(* CODESYS project base_elements.library
   Company: Vistaprint
   Version: 0.0.0.1
   Title: Base_Elements

Project tree, tasks and I/O mapping:
  libraries: Base_PLC, 0.3.2.0 (Vistaprint); Tc2_EtherCAT, 3.3.0.0 (Beckhoff Automation GmbH); Tc2_SerialCom, 3.3.0.0 (Beckhoff Automation GmbH); Tc2_Standard, * (Beckhoff Automation GmbH); Tc2_System, * (Beckhoff Automation GmbH); Tc2_Utilities, 3.3.0.0 (Beckhoff Automation GmbH); Tc3_Interfaces, * (Beckhoff Automation GmbH); Tc3_Module, * (Beckhoff Automation GmbH)
  POUs/
    Controller/
      Driver/
        RFD (RFID Driver)/
          data type E_Typ_Baudrate
          data type E_Typ_Ftim
          function block FB_Com_3964R [ST]
          function block FB_ExCom [ST]
          function FB_HEXSTRING_TO_ULINT [ST]
          function block FB_RFD [ST]: CtrlInit, CycleEndDuty, CycleStartDuty, FB_init, getCmdState, getSIf, sta_CheckBusy, sta_Error, sta_MDSBusy, sta_Off, sta_OffBusy, sta_PowerOnBusy, sta_ReadBusy, sta_SLGBusy, sta_TagInitBusy, sta_WaitForJob, sta_WriteBusy, StateMachine, StateMachine_Service
          function block FB_RFR [ST]: CtrlInit, CycleEndDuty, CycleStartDuty, FB_init, getCmdState, getSIf, sta_Error, sta_PowerOnBusy, sta_WaitForJob, StateMachine, StateMachine_Service
          global variables RFD_Cmd
          global variables RFD_Constants
          data type T_RFD
          data type T_RFD_Cfg
          data type T_RFD_Cur
          data type T_RFD_Error
          data type T_RFD_MDS_Diagnose
          data type T_RFD_MDS_State
          data type T_RFD_SLG_Diagnose
          data type T_RFD_SLG_State
          data type T_RFD_StateMachine
          data type T_RFD_Status
          data type T_StateWord
      Lvl0/
        RFW (RFID Reader-Writer)/
          data type E_Typ_RFW
          function block FB_DtChnToLine_NewRFID [ST]: Creat
          function block FB_RFW [ST]: Always, FB_init, getCmdState, getCtrlSIf, IoInBridge, IoOutBridge, sta_ERROR, sta_OFF, sta_OFFBusy, sta_PON, sta_PONBusy, sta_READ, sta_READBusy, sta_RUN, sta_RUNbusy, sta_WRITE, sta_WRITEBusy, StateMachine
          function FB_ULINT_TO_HEXSTRING [ST]
          global variables RFID_Data
          global variables RFW_CmdState
          data type T_Ctrl_SIf_RFW
          data type T_Ctrl_SIf_RFW_Cfg
          data type T_Ctrl_SIf_RFW_Cur
          data type T_Ctrl_SIf_RFW_DtChnToLine
          data type T_Ctrl_SIf_RFW_In
          data type T_Ctrl_SIf_RFW_Out
          data type T_Ctrl_SIf_RFW_Par
          data type T_NewRFID_DtChn
          data type T_RFW
      Lvl1/
      Lvl2/
      Lvl3/
    Utility Functions/
  Version/
    global variables Global_Version
*)

// POUs/Controller/Driver/RFD (RFID Driver)/E_Typ_Baudrate
TYPE E_Typ_Baudrate :
(
	baud_2400 := 4,
	baud_4800 := 5,
	baud_9600 := 6,
	baud_19200 := 7,
	baud_38400 := 8,
	baud_57600 := 9,
	baud_115200 := 10
);
END_TYPE

// POUs/Controller/Driver/RFD (RFID Driver)/E_Typ_Ftim
TYPE E_Typ_Ftim :
(
	/// Setting for air interface
	RF300 := 0,
	ISO_generall := 1,
	ISO_infineon := 3,
	ISO_Fujitsu := 4,
	ISO_NXP := 5,
	ISO_TI := 6,
	ISO_ST := 7,
	Max_E_Typ_Ftim
);
END_TYPE

// POUs/Controller/Driver/RFD (RFID Driver)/T_RFD
TYPE T_RFD :
STRUCT
	strState: STRING;
	strCmd: STRING;
	intCmd: INT;
	intServiceCmd: INT;
	stStatus: T_RFD_Status;
	stCfg: T_RFD_Cfg;
	stCur: T_RFD_Cur;
	stErr: T_RFD_Error;
END_STRUCT
END_TYPE

// POUs/Controller/Driver/RFD (RFID Driver)/T_RFD_Cfg
TYPE T_RFD_Cfg :
STRUCT
	bolSimulation: BOOL;
	eTyp: E_Typ_RFW;
	/// Reset parameter value
	usiResetParameter: USINT := 2#101010;
	/// Setting of the Air interface
	usiFtimSetting: E_Typ_Ftim;
	/// Reset option1 value
	usiResetOption1: USINT := 2#10;
	/// Set Baudrate
	uinBaudrate: USINT;
	/// Set Communikationsettings
	uinComSettings: USINT;
	/// Net ID oft EtherCat Master
	stNetId: TC2_SYSTEM.T_AmsNetID;
	/// Port Number of EtherCat Slave Comunication Module
	uinSlaveAddr: UINT;
	/// CoE Object Index for Communication Settings
	uinCoeIndexComSettings: WORD := 16#8000;
	/// CoE Object SubIndex for Baudrate
	usiCoeSubindexComBaudrate: BYTE := 16#11;
	/// CoE Object SubIndex for Dataframe
	usiCoeSubindexComDataframe: BYTE := 16#15;
	/// Retry Job to RFID Reader
	udiRetry: UDINT := 10;
	//////////////////////////////////////////////////
	/// Reset Memory 00=RAM, 01=remanent
	usiMemory: USINT := 0;
	/// Scan Mode 00= Continous Read; 01=Single Read
	usiScanMode: USINT := 1;
	/// Lock Time in ms
	uinLockTime_ms: UINT := 5000;
END_STRUCT
END_TYPE

// POUs/Controller/Driver/RFD (RFID Driver)/T_RFD_Cur
TYPE T_RFD_Cur :
STRUCT
	/// Pointer to Received Data Array
	pData: POINTER TO ARRAY[0..255] OF BYTE;
	/// Startadress to Read/Write at the data Array Element
	uinAdressData: UINT;
	/// Startadress to Read/Write at the Tag
	uinAdressTag: UINT;
	/// Number of bytes to Read/Write
	usiCount: USINT;
END_STRUCT
END_TYPE

// POUs/Controller/Driver/RFD (RFID Driver)/T_RFD_Error
TYPE T_RFD_Error :
STRUCT
	/// Reset failure
	bolErrAck: BOOL;
	/// atleast one failure active
	bolErrorActive: BOOL;
	/// error at communication card
	bolComError: BOOL;
	bolProtcolError: BOOL;
	/// Error with RF ID Tag
	bolRFIDError: BOOL;
	/// Error at setting of the communication Card (SDO Write)
	bolSDOError: BOOL;
	/// information to Communication Card error
	udiErrorID: UDINT;
END_STRUCT
END_TYPE

// POUs/Controller/Driver/RFD (RFID Driver)/T_RFD_MDS_Diagnose
TYPE T_RFD_MDS_Diagnose :
STRUCT
	/// Power flux density: as smaller the value, as higher the field intensity
	usiLFD: USINT;
	/// Errorcounter inactive mode
	usiFZP: USINT;
	/// Errorcounter active: CRC or signature errors
	usiFZA: USINT;
	/// Presence time of tag, resolution in 9.7ms
	usiANWZ: USINT;
END_STRUCT
END_TYPE

// POUs/Controller/Driver/RFD (RFID Driver)/T_RFD_MDS_State
TYPE T_RFD_MDS_State :
STRUCT
	/// MDS Type 1=no FRAM; 2=8k FRAM; 3=32k FRAM; 4=64k FRAM; 5=128k FRAM; 6=256k FRAM
	bytMDSType: BYTE;
	/// Lock bit registers (lock state)
	bytLockState: BYTE;
	/// MDS Version
	bytVersion: BYTE;
	/// Memory Size
	worMemSize: WORD;
	/// Blocksize in Byte
	bytBlockSize: BYTE;
	/// Value of memory Blocks
	bytBlockNo: BYTE;
END_STRUCT
END_TYPE

// POUs/Controller/Driver/RFD (RFID Driver)/T_RFD_SLG_Diagnose
TYPE T_RFD_SLG_Diagnose :
STRUCT
	/// Mode SLG Diagnose
	usiS_Info: USINT;
	/// Errorcounter inactive mode
	usiFZP: USINT;
	/// Counter abort
	usiABZ: USINT;
	/// Errorcounter code errors
	usiCFZ: USINT;
	/// Errorcounter signature errors
	usiSFZ: USINT;
	/// Errorcounter CRC
	usiCRCFZ: USINT;
	/// Actual command state
	usiBSTAT: USINT;
	/// Counter interface errors to host (Parity, BCC, Frame)
	usiASMFZ: USINT;
END_STRUCT
END_TYPE

// POUs/Controller/Driver/RFD (RFID Driver)/T_RFD_SLG_State
TYPE T_RFD_SLG_State :
STRUCT
	/// HW Type of SLG  0=RF310R RF340R RF350R (-xAA10); 1=RF380R (-3AA10); 2=RF310R(-1AB10); 3=RF380R (-3AB10); 4=RF340R RF350R (-2AB10,-4AB10)
	bytHWType: BYTE;
	/// HW Version
	worHWVersion: WORD;
	/// Loading Version
	worURLVersion: WORD;
	/// FW Type
	bytFWType: BYTE;
	/// FW Version
	worFWVersion: WORD;
	/// Driver Type 1=3964R
	bytDriverType: BYTE;
	/// Driver Version
	worDriverVersion: WORD;
	/// Communication port 1=RS422, 2=RS232
	bytComm: BYTE;
	/// Communication Baud rate 1=19.2kBaud; 3=57.6kBaud; 5=115.2kBaud
	bytBaud: BYTE;
	/// sending power (only RF380R) 0=standard; 2=0.5W; 3=0.75W; 4=1W; 5=1.25W (default); 6=1.5W; 7=1.75W; 8=2W
	bytPower: BYTE;
	/// Number of maximal tags in the field
	bytMtag: BYTE;
	/// air interface 0=RF300; 1=ISO generall; 3=ISO infineon Chip; 4=ISO Fujitsu; 5=ISO NXP; 6=ISO TI; 7=ISO ST
	bytFtim: BYTE;
	/// State antenna 1=ON; 2=OFF
	bytAntenna: BYTE;
	/// Tag presence 0=No presence; 1=prexence
	bytPresence: BYTE;
END_STRUCT
END_TYPE

// POUs/Controller/Driver/RFD (RFID Driver)/T_RFD_StateMachine
TYPE T_RFD_StateMachine :
STRUCT
	///actual state
	intState: INT;
	///state of last cycle
	intStateLastCycle: INT;
	///save history backup p.e. in ERROR state
	intStateHistory: INT;
	///set state for next cycle
	intStateNext: INT;
	///Time in this State
	udiTimeInState_ms: UDINT;
END_STRUCT
END_TYPE

// POUs/Controller/Driver/RFD (RFID Driver)/T_RFD_Status
TYPE T_RFD_Status :
STRUCT
	/// 1 = Antenna is initialized  
	bolStartupOk: BOOL;
	/// 1 = Antenna is initialized  
	bolInitOk: BOOL;
	/// 1 = Antenna is on 
	bolOn: BOOL;
	/// 1 = tag is present  
	bolPresent: BOOL;
	/// 1 = Communication to SLG is OK  
	bolL_UEB: BOOL;
	/// SLG State only actual on demand 
	stSLG_State: T_RFD_SLG_State;
	/// SLG Diagnose only actual on demand 
	stSLG_Diag: T_RFD_SLG_Diagnose;
	/// SLG State only actual on demand  
	stMDS_State: T_RFD_MDS_State;
	/// SLG Diagnose only actual on demand  
	stMDS_Diag: T_RFD_MDS_Diagnose;
	/// Tag ID
	abyteUID: ARRAY[0..7] OF BYTE;
END_STRUCT
END_TYPE

// POUs/Controller/Driver/RFD (RFID Driver)/T_StateWord
TYPE T_StateWord :
STRUCT
	///Acknowledge the datachange of this Command bit
	bolTransmitAccepted: BOOL;
	///New Datat at the input
	bolReceiveRequest: BOOL;
	///0=Ready for Data exchange; 1=initialisation of the clam
	bolInputAccepted: BOOL;
	///Input Buffer is full, all new arriveing data lost
	bolBufferFull: BOOL;
	///Parity Error occured
	bolParityErr: BOOL;
	///Framing Error occured
	bolFramingErr: BOOL;
	///Overrun Error occured
	bolOverrunErr: BOOL;
	///Amounth of the reached Input Bytes
	usiInLenght: USINT;
END_STRUCT
END_TYPE

// POUs/Controller/Lvl0/RFW (RFID Reader-Writer)/E_Typ_RFW
TYPE E_Typ_RFW :
(
	/// RF310
	RF310R := 0,
	/// RF382R
	RF382R := 1,
	Max_E_Typ_CYL
);
END_TYPE

// POUs/Controller/Lvl0/RFW (RFID Reader-Writer)/T_Ctrl_SIf_RFW
TYPE T_Ctrl_SIf_RFW :
STRUCT
	///configuration
	Cfg: T_Ctrl_SIf_RFW_Cfg;
	///parameter
	Par: T_Ctrl_SIf_RFW_Par;
	///current values
	Cur: T_Ctrl_SIf_RFW_Cur;
	///io input
	In: T_Ctrl_SIf_RFW_In;
	///io output
	Out: T_Ctrl_SIf_RFW_Out;
	///alarm number used in this controller
	Alm: ARRAY[1..5] OF T_Ctrl_Alm;
END_STRUCT
END_TYPE

// POUs/Controller/Lvl0/RFW (RFID Reader-Writer)/T_Ctrl_SIf_RFW_Cfg
TYPE T_Ctrl_SIf_RFW_Cfg :
STRUCT
	eTyp: E_Typ_RFW;
	/// Get automatically the Tray ID too 
	bolGetTrayIDAuto: BOOL;
	/// Net ID oft EtherCat Master
	stNetId: TC2_SYSTEM.T_AmsNetID;
	/// Port Number of EtherCat Slave Comunication Module
	uinSlaveAddr: UINT;
END_STRUCT
END_TYPE

// POUs/Controller/Lvl0/RFW (RFID Reader-Writer)/T_Ctrl_SIf_RFW_Cur
TYPE T_Ctrl_SIf_RFW_Cur :
STRUCT
	/// 1 = tag is present  
	bolPresent: BOOL;
	/// Data to read / write
	abytData: ARRAY[0..255] OF BYTE;
	/// Data in Structure
	stData: T_RFW;
	/// Job information, what data read or write
	dwoJob: DWORD;
END_STRUCT
END_TYPE

// POUs/Controller/Lvl0/RFW (RFID Reader-Writer)/T_Ctrl_SIf_RFW_DtChnToLine
TYPE T_Ctrl_SIf_RFW_DtChnToLine :
STRUCT
	stNewRfid: T_NewRFID_DtChn;
END_STRUCT
END_TYPE

// POUs/Controller/Lvl0/RFW (RFID Reader-Writer)/T_Ctrl_SIf_RFW_In
TYPE T_Ctrl_SIf_RFW_In :
STRUCT
END_STRUCT
END_TYPE

// POUs/Controller/Lvl0/RFW (RFID Reader-Writer)/T_Ctrl_SIf_RFW_Out
TYPE T_Ctrl_SIf_RFW_Out :
STRUCT
END_STRUCT
END_TYPE

// POUs/Controller/Lvl0/RFW (RFID Reader-Writer)/T_Ctrl_SIf_RFW_Par
TYPE T_Ctrl_SIf_RFW_Par :
STRUCT
	///[ms] until failure to long time for read
	udiReadTime_ms: UDINT;
	///[ms] until failure to long time for write
	udiWriteTime_ms: UDINT;
END_STRUCT
END_TYPE

// POUs/Controller/Lvl0/RFW (RFID Reader-Writer)/T_NewRFID_DtChn
TYPE T_NewRFID_DtChn :
STRUCT
	// new RF ID
	strID: STRING;			// configurable if Tag or Tray ID
	uliTagID: ULINT;
	dtTimestamp: DT;
	intDataState: INT;	
END_STRUCT
END_TYPE

// POUs/Controller/Lvl0/RFW (RFID Reader-Writer)/T_RFW
TYPE T_RFW :
STRUCT
	///	Repeteition ID			Identifies the try number in the sequence	
	usiRepetitionID: USINT;
	///	Workstation		2 workstations in the cell	1 BIT	0: Workstation1, 2: Workstation2
	bolWorkstation2: BOOL;
	///usiProductID : USINT;				// 	The product ID bits 1 to 5 are indeed not used. Mail T.Bosgiraud 11.6.2013 Product type	Max number of product types = 32	5 bits,	product ID (bits 1 to 5), 
	bolDeleteFileAfterPrint: BOOL;
	/// 	1 means that the image has been printed without problem.
	bolPrintOk: BOOL;
	///	0: Use the bottom of the tray as basis and add Offset
	bolHeightUseMeasure: BOOL;
	///	Email 1.06.2013 Berk “Use measured height=1”, the actual measurement of the  laser plus any offsets programmed into the tray are used to adjust the lifting height
	///	1: Use the printable product surface as basis and add Offset to the measured height
	usiHeightOffset: USINT;
	/// 	“Offset +/-” = 1 means that the printable surface OF the item will go further away FROM the print head.
	bolHeightOffsetSignMinus: BOOL;
	/// 	“Offset +/-” = 0 (default value) means that the printable surface of the item will come closer to the print head
	bolIonizer: BOOL;
	/// 	Pre-treatment	Plasma 0: Plasma off, 1: Level 1 ..3:Level3
	usiPlasmaLevel: USINT;
	/// 	Print numbers 1 means that the image needs to be printed twice on the products
	bolPrintPass: BOOL;
	/// 	1 means that the nozzle check pattern has to be printed onto the products.
	bolNozzleCheck: BOOL;
	///	1 means that the alignment check pattern has to be printed onto the products.
	bolAligneCheck: BOOL;
	///	UV-pinning intensity 0: Level1 ... 15: Level16
	usiUVPinningLevel: USINT;
	///	UV-lamp intensity 0: Level1 ... 15: Level16
	usiUVLampLevel: USINT;
	/// p.e.: 268205625-3.pdf -> The file name sent by VIPER to the printer and to the conveyor is made out of 64 bits
	strFileName: STRING;
	/// The RFID divides the rest of the name (268205625-3) as 8 successive bytes arranged as follows:
	///	-	Byte 7 (RFID byte 0Dhex) to byte 1 (RFID byte 07hex) express the number before the hyphen sign (in this case 268205625)
	///	-	Byte 0 (RFID byte 06hex) expresses the number after the hyphen sign (in this case 3).
	bolBrush: BOOL;
	///	1: use second brush means that the brush has TO be used FOR the considered tray
	bolBrushClean: BOOL;
	///	“Brush Fans”=1 means that the fans have to be used for the considered tray
	bolBrushFans: BOOL;
	///	“Gutter Clean”=1 means that the tray is running for gutter cleaning purposes.
	bolGutterClean: BOOL;
	/// 	This bit tells whether the tray is a regular production tray or a special tray (nozzle check, alignment...).
	bolSpecialTray: BOOL;
	/// 	Byte 0-13	->9999999999999	
	strTrayID: STRING;
	/// 	Byte 0-13	->9999999999999	
	strTagID: STRING;
	uliTagID: ULINT;
END_STRUCT
END_TYPE

// POUs/Controller/Driver/RFD (RFID Driver)/RFD_Cmd
VAR_GLOBAL CONSTANT
	/// ctrl state definitions
	/// Error
	cRFD_STA_Error: INT := 256;
	/// Power On
	cRFD_STA_PowerOnBusy: INT := 999;
	cRFD_STA_WaitForJob: INT := 1002;
	/// RESET Reader 
	cRFD_STA_ResetBusy: INT := 1003;
	/// Turn Off antenna 
	cRFD_STA_OffBusy: INT := 1007;
	cRFD_STA_Off: INT := 1008;
	/// Write Data to Tag 
	cRFD_STA_WriteBusy: INT := 1009;
	/// Read Data from Tag 
	cRFD_STA_ReadBusy: INT := 1011;
	/// Tag initialisation 
	cRFD_STA_TagInitBusy: INT := 1013;
	/// Check connection to antenna
	cRFD_STA_CheckBusy: INT := 1017;
	/// Service function read MDS-State (State of the near Tag)
	cRFD_STA_MDSBusy: INT := 1019;
	/// Service function read SLG State (State of the antenna)
	cRFD_STA_SLGBusy: INT := 1021;
	/// ctrl commands definitions
	/// specific commands >200 - every command has to be a even number
	cRFD_CMD_DONE: INT := -1;
	/// Switch controller on 
	cRFD_CMD_CTRL_ON: INT := 1000;
	/// Switch controller off 
	cRFD_CMD_CTRL_OFF: INT := 1006;
	/// Write Data to Tag 
	cRFD_CMD_Write: INT := 1010;
	/// Read Data from Tag 
	cRFD_CMD_Read: INT := 1012;
	/// Check connection to antenna 
	cRFD_CMD_Check: INT := 1018;
	/// Service function read MDS-State (State of the near Tag)
	cRFD_CMD_MDS: INT := 1020;
	/// Service function read SLG State (State of the antenna)
	cRFD_CMD_SLG: INT := 1022;
	/// Sub States
	/// Power On Busy
	cRFD_SUB_SetBaudrate: INT := 2001;
	/// Set Communication Settings
	cRFD_SUB_SetComSettings: INT := 2002;
	///  Clear Buffer
	cRFD_SUB_ClearBuffer: INT := 2003;
	/// Initialisation String sending
	cRFD_SUB_InitString: INT := 2004;
	///  Check Power On State
	cRFD_SUB_CheckPon: INT := 2005;
	/// OFF Busy
	cRFD_SUB_Prepare: INT := 2010;
	/// Data send
	cRFD_SUB_SendBusy: INT := 2011;
	/// Wait Answer
	cRFD_SUB_WaitAnswer: INT := 2012;
	/// SLG Write Mode 1
	cRFD_SUB_Write1: INT := 2020;
	/// SLG Wait Mode 1
	cRFD_SUB_Wait1: INT := 2021;
	/// SLG Write Mode 6
	cRFD_SUB_Write6: INT := 2022;
	/// SLG Wait Mode 6
	cRFD_SUB_Wait6: INT := 2023;
	///  Substates finished
	cRFD_SUB_SubStatesEnd: INT := 2100;
END_VAR

// POUs/Controller/Driver/RFD (RFID Driver)/RFD_Constants
VAR_GLOBAL
END_VAR

// POUs/Controller/Lvl0/RFW (RFID Reader-Writer)/RFID_Data
VAR_GLOBAL CONSTANT
	/// RFID Data connection
	/// See RFID Specification
	/// Defines the Start Adress and the lengh of the Data in the RF ID Tag
	/// Every DoubleWord has to Words, Higher is lengh, lower word is Startadress
	/// Example	
	/// 16#010005 => Startadress 5 Byte 1 => UV Settings
	cRFID_RepetionID: DWORD := 16#10101;
	cRFID_TrayInfo: DWORD := 16#10102;
	cRFID_HeighOfTray: DWORD := 16#10103;
	cRFID_Pretreatment: DWORD := 16#10104;
	cRFID_UVcuring: DWORD := 16#10105;
	cRFID_Filename: DWORD := 16#80106;
	cRFID_Brush: DWORD := 16#1010E;
	cRFID_TrayID: DWORD := 16#E0000;
	cRFID_TagID: DWORD := 16#8FFF0;
	cRFID_AllData: DWORD := 16#F0100;
END_VAR

// POUs/Controller/Lvl0/RFW (RFID Reader-Writer)/RFW_CmdState
VAR_GLOBAL CONSTANT
	///ctrl commands definitions
	///specific commands >200 - every command has to be a even number
	cCMD_READ: INT := 202;
	cCMD_WRITE: INT := 204;
	///ctrl specific states definitions
	cSTA_READBusy: INT := 201;
	cSTA_READ: INT := cCMD_READ;
	cSTA_WRITEBusy: INT := 203;
	cSTA_WRITE: INT := cCMD_WRITE;
END_VAR

// Version/Global_Version
// This function has been automatically generated from the project information.
VAR_GLOBAL CONSTANT
	{attribute 'const_non_replaced'}
	stLibVersion_Base_Elements : ST_LibVersion := (iMajor := 0, iMinor := 0, iBuild := 0, iRevision := 1, sVersion := '0.0.0.1');
END_VAR

// POUs/Controller/Driver/RFD (RFID Driver)/FB_Com_3964R
FUNCTION_BLOCK FB_Com_3964R
VAR_INPUT
	/// Pointer to Received Data Array
	In_pRxData: POINTER TO ARRAY[0..255] OF BYTE;
	/// Pointer to Sending Data Array
	In_pTxData: POINTER TO ARRAY[0..255] OF BYTE;
	/// Amounth of sending data
	In_udiTxCount: UDINT;
	/// Error Acknowledge 
	In_bolErrorAck: BOOL;
END_VAR
VAR_IN_OUT
	/// Command to send Data 1=command; 0=Done
	InOut_bolSend: BOOL;
	/// Command Data received 1=received; 0=Done=Ready for next Data
	InOut_bolRec: BOOL;
END_VAR
VAR_OUTPUT
	/// Amounth of received data
	Out_udiRxCount: UDINT;
	/// Serial interface communication error
	Out_bolComError: BOOL;
	/// Error in protocoll procedure
	Out_bolProtocolErr: BOOL;
	/// Error information to master
	Out_udiErrorCode: UDINT;
END_VAR
VAR
	In_stEL6inData AT %I*: TC2_SERIALCOM.EL6inData22B;
	Out_stEL6outData AT %Q*: TC2_SERIALCOM.EL6outData22B;
	/// Internal Variables
	udiI: UDINT;
	/// Local variable for loops
	udiK: UDINT;
	/// Internal Error Reset
	bolIntReset: BOOL;
	/// Count call trials
	uinCountCall: UINT;
	/// Count call Retrys
	uinCountRetry: UINT;
	/// Temporary value for cecking the sum
	bytCheckValue: BYTE;
	/// Antenna is initializied, until it is not initializied, it send 16#02 in all possible baudrates
	bolSLGInitialized: BOOL := FALSE;
	/// Check Timeout
	bolTimeout: BOOL;
	/// Check Timeout
	bolWait: BOOL;
	/// Send NAK needed
	bolSendNAK: BOOL;
	/// Receive Wait signs
	timWaitReceive: TIME := TIME#5ms;
	/// Receive Wait signs
	timWaitAck: TIME := TIME#400ms;
	/// Sign delay time
	timZVZ: TIME := TIME#45ms;
	/// Time ACK delay
	timQVZ: TIME := TIME#145ms;
	/// Initialisation of the HW card
	bolInitRequest: BOOL;
	/// Setting of the HW Card
	bolSendContinious: BOOL;
	/// Priority at RFID
	bolPriority: BOOL;
	/// Send DLE doubletimes
	bolDLEDouble: BOOL;
	/// New data received
	bolComDataReceived: BOOL;
	/// receiving busy
	bolComRecBusy: BOOL;
	/// Received Data
	udiComSizeReceiveData: UDINT;
	/// Sending busy
	bolComSendBusy: BOOL;
	/// Error at serial line control
	bolErrSerialLineControl: BOOL;
	/// Error at serial line control
	stErrSerialLineControl: ComError_t;
	/// Error at serial line  receiving data
	bolErrReceive: BOOL;
	/// Error at serial line  receiving data
	stErrReceive: ComError_t;
	/// Error at serial line sending data
	bolErrSend: BOOL;
	/// Error at serial line sending data
	stErrSend: ComError_t;
	/// Define Buffer for preparations
	aRxData: ARRAY[0..255] OF BYTE;
	aTxData: ARRAY[0..255] OF BYTE;
	/// Define Buffer for Funciton
	stRxBuffer: TC2_SERIALCOM.ComBuffer;
	/// Transmit data buffer; used with all receive function blocks 
	stTxBuffer: TC2_SERIALCOM.ComBuffer;
	/// Sub Statemachine
	intState: INT := 0;
	intStateOld: INT := 0;
	udiStateLoop: UDINT;
	a_intStateHist: ARRAY[0..9] OF INT;
	udiStateDebug: UDINT;
	udiStateDebugMax: UDINT;
	/// Function for serial communication
	fbSerialLineControl: TC2_SERIALCOM.SerialLineControl;
	fbSerialReceiveData: TC2_SERIALCOM.ReceiveData;
	fbSerialSendData: TC2_SERIALCOM.SendData;
	fbSerialClearComBuffer: TC2_SERIALCOM.ClearComBuffer;
	fbTon: TC2_STANDARD.TON;
	fbWait: TC2_STANDARD.TON;
	fbZVZ: TC2_STANDARD.TON;
	fbQVZ: TC2_STANDARD.TON;
	fbPriority: TC2_STANDARD.TON;
END_VAR
VAR CONSTANT
	cSTX: USINT := 16#2;
	cDLE: USINT := 16#10;
	cETX: USINT := 16#3;
	cNAK: USINT := 16#15;
	/// Startup
	cRFD_3964_Start: INT := 2500;
	/// Startup
	cRFD_3964_Init: INT := 2501;
	/// Wait for Job
	cRFD_3964_Wait: INT := 2502;
	/// Read recived sign
	cRFD_3964_RxRead: INT := 2504;
	/// Ackn. receiving ready
	cRFD_3964_RxReadRdy: INT := 2506;
	/// Recive Data
	cRFD_3964_RxData: INT := 2508;
	/// Achn. received Data
	cRFD_3964_RxCheckData: INT := 2510;
	/// Send Ack to Slave
	cRFD_3964_RxAck: INT := 2512;
	/// Send Ack to Slave
	cRFD_3964_RxAck2: INT := 2514;
	/// Send Request to Slave
	cRFD_3964_TxRequest: INT := 2550;
	/// Send Wait answer
	cRFD_3964_TxWait: INT := 2552;
	/// Send Data
	cRFD_3964_TxSend: INT := 2554;
	/// Send Wait for Ack
	cRFD_3964_TxAck: INT := 2556;
	/// Error
	cRFD_3964_Error: INT := 2580;
END_VAR

(*__________________________________________________________________________________________________
¦	
¦	Vistaprint Schweiz GmbH
¦	CH - 8401 Winterthur
¦
¦	www.vistaprint.ch - info@vistaprint.ch
¦___________________________________________________________________________________________________

Function desription:
Driver for communication protocoll 3964R
Description in Siemens manual from CP341, A5E02191070-03


History:
Version		Date			Author		Comment
---------------------------------------------------------------------------------------------------
0.00.1		23.07.2013		AVME/PRE	Start history
___________________________________________________________________________________________________*)

// Always
fbSerialLineControl(
	Mode:= TC2_SERIALCOM.ComSerialLineMode_t.SERIALLINEMODE_EL6_22B, 
	pComIn:= ADR(In_stEL6inData), 
	pComOut:= ADR(Out_stEL6outData), 
	SizeComIn:= SIZEOF(In_stEL6inData), 
	Error=> bolErrSerialLineControl, 
	ErrorID=> stErrSerialLineControl, 
	TxBuffer:= stTxBuffer, 
	RxBuffer:= stRxBuffer);
	
// Check timers
IF intState >= cRFD_3964_Wait THEN
	fbZVZ(PT:= timZVZ);
	fbQVZ(PT:= timQVZ);
	fbWait(PT:= timWaitAck);

	// Check priority
	fbPriority(IN:= bolPriority, PT:=timWaitAck);
	IF (fbPriority.Q = TRUE) THEN
		bolPriority := FALSE;
	END_IF

END_IF
		
// Startup set correct Step
IF intState < cRFD_3964_Start THEN
	intState := cRFD_3964_Start;
END_IF

// State Machine
CASE intState OF
	cRFD_3964_Start:
		// Clear Buffer
		FOR udiI := 0 TO SIZEOF(aRxData)-1 DO
			aRxData[udiI] := 0;
			aTxData[udiI] := 0;
		END_FOR
		bolSLGInitialized := FALSE;
		
		// Clear counters
		uinCountCall := 0;
		uinCountRetry := 0;
		
		bolInitRequest := FALSE;
		bolSendContinious := FALSE;
		
		
		// Next State
		IF (bolErrSerialLineControl = FALSE) AND (bolTimeout=TRUE) THEN
			intState := cRFD_3964_Init;
		ELSIF (bolErrSerialLineControl = TRUE) THEN
			intState := cRFD_3964_Error;
		END_IF

	// Wait for a job or received Data //	
	cRFD_3964_Init:	
		bolInitRequest := TRUE;
		
		IF (bolErrSerialLineControl = FALSE) AND ((In_stEL6inData.Status.2 = TRUE) OR (bolTimeout=TRUE)) THEN	// Initialisation Done  OR (bolTimeout=TRUE)
			intState := cRFD_3964_Wait;
		ELSIF (bolErrSerialLineControl = TRUE) THEN
			intState := cRFD_3964_Error;
		END_IF
	
	// Wait for a job or received Data //	
	cRFD_3964_Wait:	
		bolInitRequest := FALSE;
		bolSendNAK := FALSE;
		fbZVZ.IN := FALSE;
		fbQVZ.IN := FALSE;
		fbWait.IN := FALSE;
		
		fbSerialReceiveData(
		//	pPrefix:= , // Not used because no prefix in telegram
			LenPrefix:= 0, 
		//	pSuffix:= , // Not used because no suffix in telegram
			LenSuffix:= 0, 
			pReceiveData:= ADR(aRxData), 
			SizeReceiveData:= 255, 
			Timeout:= timWaitReceive, 
		//	Reset:= , 
			DataReceived=> bolComDataReceived, 
			busy=> bolComRecBusy, 
			Error=> stErrReceive, 
			RxTimeout=> bolErrReceive, 
			LenReceiveData=> udiComSizeReceiveData, 
			RXbuffer:= stRxBuffer);
		
		//Check if Data is received
		IF bolComDataReceived = TRUE THEN
			intState := cRFD_3964_RxRead;
		ELSIF (InOut_bolSend = TRUE) AND (bolPriority = FALSE) THEN
			intState := cRFD_3964_TxRequest;
		END_IF
			
	// Read first signs if new data sending needed //	
	cRFD_3964_RxRead: 
		// Check reached Sign
		// Send ready for reach Data if STX is send and Buffer is ready to use
		fbWait.IN := TRUE;
		IF (((aRxData[0] = cSTX) OR (bolSLGInitialized = FALSE))  AND (InOut_bolRec = FALSE)) THEN 
			aTxData[0] := cDLE;
		ELSE
			aTxData[0] := cNAK;
		END_IF
		
		IF ((fbWait.Q = FALSE) OR (InOut_bolRec = TRUE)) THEN
			intState := cRFD_3964_RxReadRdy; 
			fbWait.IN := FALSE; 
		END_IF
		
	// Send Feedback //		
	cRFD_3964_RxReadRdy:
		fbZVZ.IN := TRUE; 

		IF fbZVZ.Q = TRUE THEN
			fbSerialSendData(
				pSendData:= ADR(aTxData), 
				Length:= 1, 
				Busy=> bolComSendBusy, 
				Error=> stErrSend, 
				TXbuffer:= stTxBuffer);
				bolSendContinious := TRUE;
		END_IF
			
		// Check transition
		IF (bolComSendBusy = FALSE) AND (bolSLGInitialized = TRUE) AND (fbZVZ.Q = TRUE) THEN		// AND (stErrSend = 0)
			IF (aTxData[0] = cDLE) THEN
				intState := cRFD_3964_RxData;
			ELSE
				intState := cRFD_3964_Wait;
			END_IF
		ELSIF ((bolComSendBusy = TRUE) OR (bolTimeout = TRUE)) AND (uinCountCall < 10) AND (fbZVZ.Q = TRUE) THEN
			uinCountCall := uinCountCall + 1;
			intState := cRFD_3964_Wait;
		ELSIF ((bolComSendBusy = TRUE) OR (bolTimeout = TRUE)) AND (fbZVZ.Q = TRUE) THEN
			bolSendNAK := TRUE;
			intState := cRFD_3964_Error;
		END_IF
		
	// Read Data //	
	cRFD_3964_RxData:
		fbZVZ.IN := FALSE; 
		fbSerialReceiveData(
		//	pPrefix:= , // Not used because no prefix in telegram
			LenPrefix:= 0, 
		//	pSuffix:= , // Not used because no suffix in telegram
			LenSuffix:= 0, 
			pReceiveData:= ADR(aRxData), 
			SizeReceiveData:= 255, 
			Timeout:= timWaitReceive, 
		//	Reset:= , 
			DataReceived=> bolComDataReceived, 
			busy=> bolComRecBusy, 
			Error=> stErrReceive, 
			RxTimeout=> bolErrReceive, 
			LenReceiveData=> udiComSizeReceiveData, 
			RXbuffer:= stRxBuffer);
				
		IF (bolComDataReceived = TRUE) AND (bolComRecBusy = FALSE) AND (udiComSizeReceiveData <= 255)  THEN
			intState := cRFD_3964_RxCheckData;
		ELSIF ((bolTimeout = TRUE) OR (udiComSizeReceiveData > 255)) THEN	 // OR (stErrReceive <> 0)
			bolSendNAK := TRUE;
			IF (uinCountCall < 10) THEN
				uinCountCall := uinCountCall + 1;
				intState := cRFD_3964_RxAck;
			ELSE
				intState := cRFD_3964_Error;
			END_IF
		END_IF
	
	// Check Received Data //	
	cRFD_3964_RxCheckData:
		//minimal 1 Byte, ETX and BCC   	ETX is last sign for BCC					DLE is last sign for ETX
		IF (udiComSizeReceiveData >= 4) THEN
			IF ((aRxData[udiComSizeReceiveData-2] = cETX) AND (aRxData[udiComSizeReceiveData-3] = cDLE)) THEN
				// Check BCC
				bytCheckValue := aRxData[0] XOR aRxData[1];
				FOR udiI := 2 TO  (udiComSizeReceiveData-2) DO
					bytCheckValue := bytCheckValue XOR aRxData[udiI];
				END_FOR
				
				IF (bytCheckValue = aRxData[udiComSizeReceiveData-1]) THEN //BCC OK
					// Copy Data
					FOR udiI := 0 TO (SIZEOF(aRxData)-1) DO
						In_pRxData^[udiI] := 0;
					END_FOR
					udiK := 0;
					FOR udiI := 0 TO udiComSizeReceiveData-4 DO
						In_pRxData^[udiK] := aRxData[udiI];
						IF (aRxData[udiI] = cDLE) AND (aRxData[udiI+1] = cDLE) THEN		// DLE Doubling, only take on DLE
							udiI := udiI+1;
						END_IF
						udiK := udiK + 1;
					END_FOR
					InOut_bolRec := TRUE;
					intState := cRFD_3964_RxAck;
				ELSE
					bolSendNAK := TRUE;				
					IF (uinCountCall < 10) THEN
						uinCountCall := uinCountCall + 1;
						intState := cRFD_3964_RxAck;
					ELSE
						intState := cRFD_3964_Error;
					END_IF
				END_IF
			ELSE
				bolSendNAK := TRUE;				
				IF (uinCountCall < 10) THEN
					uinCountCall := uinCountCall + 1;
					intState := cRFD_3964_RxAck;
				ELSE
					intState := cRFD_3964_Error;
				END_IF
			END_IF
		ELSIF aRxData[0] = cSTX THEN
			aTxData[0] := cDLE;
			intState := cRFD_3964_RxReadRdy;
		ELSE
			bolSendNAK := TRUE;				
			IF (uinCountCall < 10) THEN
				uinCountCall := uinCountCall + 1;
				intState := cRFD_3964_RxAck;
			ELSE
				intState := cRFD_3964_Error;
			END_IF
		END_IF
	// SEND Acknowledge of received Data //
	cRFD_3964_RxAck:
		IF bolSendNAK = TRUE THEN
			aTxData[0] := cNAK;
		ELSE
			aTxData[0] := cDLE;
		END_IF
		
		fbZVZ.IN := TRUE; // Prepare for send step
		fbSerialSendData(
			pSendData:= ADR(aTxData), 
			Length:= 1, 
			Busy=> bolComSendBusy, 
			Error=> stErrSend, 
			TXbuffer:= stTxBuffer);
				
					
		// Check transition
		IF (bolComSendBusy = FALSE) AND (stErrSend = 0) AND (bolSendNAK = FALSE) THEN	//  AND (fbZVZ.Q = TRUE)
			uinCountCall := 0;
			bolSLGInitialized := TRUE;
			intState := cRFD_3964_Wait;
		ELSIF (bolComSendBusy = FALSE) AND (stErrSend = 0) AND (bolSendNAK = TRUE) THEN	//  AND (fbZVZ.Q = TRUE)
			intState := cRFD_3964_Wait;
		END_IF

	// SEND Acknowledge of received Data //
	cRFD_3964_RxAck2:
		IF bolSendNAK = TRUE THEN
			aTxData[0] := cNAK;
		ELSE
			aTxData[0] := cDLE;
		END_IF
		
		fbSerialSendData(
			pSendData:= ADR(aTxData), 
			Length:= 1, 
			Busy=> bolComSendBusy, 
			Error=> stErrSend, 
			TXbuffer:= stTxBuffer);
				
		// Check transition
		IF (bolComSendBusy = FALSE) AND (stErrSend = 0) AND (bolSendNAK = FALSE) AND (bolWait = TRUE) THEN
			uinCountCall := 0;
			bolSLGInitialized := TRUE;
			intState := cRFD_3964_Wait;
		ELSIF (bolComSendBusy = FALSE) AND (stErrSend = 0) AND (bolSendNAK = TRUE) AND (bolWait = TRUE) THEN
			intState := cRFD_3964_Wait;
		ELSIF ((bolComSendBusy = TRUE) OR (bolTimeout = TRUE)) THEN
			intState := cRFD_3964_Error;
		END_IF

/////////////////////////////////////////////////////////////////////
// Sending Data
	// Request a sending job at Slave //
	cRFD_3964_TxRequest:
		aTxData[0] := cSTX;
		fbSerialSendData(
			pSendData:= ADR(aTxData), 
			Length:= 1, 
			Busy=> bolComSendBusy, 
			Error=> stErrSend, 
			TXbuffer:= stTxBuffer);
		bolSendContinious := TRUE;
			
		// Check transition
		IF (bolComSendBusy = FALSE) AND (stErrSend = 0) THEN
			intState := cRFD_3964_TxWait;
		ELSIF ((bolComSendBusy = TRUE) OR (bolTimeout = TRUE)) THEN
			intState := cRFD_3964_Error;
		END_IF
		
	// Wait for answer ready //	
	cRFD_3964_TxWait:	
		fbSerialReceiveData(
		//	pPrefix:= , // Not used because no prefix in telegram
			LenPrefix:= 0, 
		//	pSuffix:= , // Not used because no suffix in telegram
			LenSuffix:= 0, 
			pReceiveData:= ADR(aRxData), 
			SizeReceiveData:= 1, 
			Timeout:= timWaitReceive, 
		//	Reset:= , 
			DataReceived=> bolComDataReceived, 
			busy=> bolComRecBusy, 
			Error=> stErrReceive, 
			RxTimeout=> bolErrReceive, 
			LenReceiveData=> udiComSizeReceiveData, 
			RXbuffer:= stRxBuffer);
				
		IF (bolComDataReceived = TRUE) AND (bolComRecBusy = FALSE) AND (udiComSizeReceiveData <= 255)  THEN
			IF aRxData[0] = cDLE THEN
				intState := cRFD_3964_TxSend;
			ELSIF aRxData[0] = cSTX THEN	// At Start of Text 
				intState := cRFD_3964_RxRead;
				bolPriority := TRUE;
			ELSE
				IF uinCountRetry > 10 THEN
					intState := cRFD_3964_Error;
				ELSE 
					uinCountRetry := uinCountRetry + 1;
					intState := cRFD_3964_Wait;
				END_IF
			END_IF			
		ELSIF ((bolTimeout = TRUE) OR (udiComSizeReceiveData > 255)) THEN
			IF uinCountCall > 10 THEN
				intState := cRFD_3964_Error;
			ELSE
				IF bolSLGInitialized = TRUE THEN
					uinCountCall := uinCountCall + 1;
					intState := cRFD_3964_Wait;
				END_IF
			END_IF				
		END_IF
	
	// sending data //	
	cRFD_3964_TxSend:
		//only prepare data if not sending //
		IF (bolComSendBusy = FALSE) THEN
			bolDLEDouble := FALSE;
			udiI := 11;
			FOR udiI := 0 TO (SIZEOF(aTxData)-1) DO
				aTxData[udiI] := 0;
			END_FOR
			udiI := 0;
			udiK := 0;
			FOR udiK := 0 TO In_udiTxCount-1 DO
				aTxData[udiI] := In_pTxData^[udiK];
				IF aTxData[udiI] = cDLE THEN
					udiI := udiI + 1;
					aTxData[udiI] := cDLE;
					bolDLEDouble := TRUE;
				END_IF
				udiI := udiI + 1;				
			END_FOR
			aTxData[udiI] := cDLE;
			udiI := udiI + 1;
			//IF bolDLEDouble = TRUE THEN		// DLE Doubling at the end of the data if once uced as data
			//	aTxData[udiI] := cDLE;
			//	udiI := udiI + 1;				
			//END_IF
			aTxData[udiI] := cETX;
			
			bytCheckValue := aTxData[0] XOR aTxData[1];
			FOR udiK := 2 TO  udiI DO
				bytCheckValue := bytCheckValue XOR aTxData[udiK];
			END_FOR
			udiI := udiI + 1;
			aTxData[udiI] := bytCheckValue;
			udiI := udiI + 1;
		END_IF

		fbSerialSendData(
			pSendData:= ADR(aTxData), 
			Length:= udiI, 
			Busy=> bolComSendBusy, 
			Error=> stErrSend, 
			TXbuffer:= stTxBuffer);
			
		// Check transition
		IF (bolComSendBusy = FALSE) AND (stErrSend = 0) THEN
			intState := cRFD_3964_TxAck;
		ELSIF ((bolComSendBusy = TRUE) OR (bolTimeout = TRUE)) THEN
			IF uinCountRetry > 10 THEN
				intState := cRFD_3964_Error;
			ELSE 
				uinCountRetry := uinCountRetry + 1;
				intState := cRFD_3964_Wait;
			END_IF
		END_IF
		
	// Wait for answer ready //	
	cRFD_3964_TxAck:
		fbSerialReceiveData(
		//	pPrefix:= , // Not used because no prefix in telegram
			LenPrefix:= 0, 
		//	pSuffix:= , // Not used because no suffix in telegram
			LenSuffix:= 0, 
			pReceiveData:= ADR(aRxData), 
			SizeReceiveData:= 255, 
			Timeout:= timWaitReceive, 
		//	Reset:= , 
			DataReceived=> bolComDataReceived, 
			busy=> bolComRecBusy, 
			Error=> stErrReceive, 
			RxTimeout=> bolErrReceive, 
			LenReceiveData=> udiComSizeReceiveData, 
			RXbuffer:= stRxBuffer);
				
		IF (bolComDataReceived = TRUE) AND (bolComRecBusy = FALSE) AND (udiComSizeReceiveData <= 255)  THEN
			IF aRxData[0] = cDLE THEN
				intState := cRFD_3964_Wait;
				InOut_bolSend := FALSE;
				bolSLGInitialized := TRUE;
			ELSE
				IF uinCountRetry > 10 THEN
					intState := cRFD_3964_Error;
				ELSE 
					uinCountRetry := uinCountRetry + 1;
					intState := cRFD_3964_Wait;
				END_IF
			END_IF			
		ELSIF ((bolTimeout = TRUE) OR (udiComSizeReceiveData > 255)) THEN	 // OR (stErrReceive <> 0)
			IF uinCountRetry > 10 THEN
				intState := cRFD_3964_Error;
			ELSE
				uinCountRetry := uinCountRetry + 1;
				intState := cRFD_3964_Wait;
			END_IF				
		END_IF
	

////////////////////////////////////////////////////////////		
		// Error State //
		cRFD_3964_Error:
			// Send correct information
			IF bolErrSerialLineControl = TRUE THEN
				Out_udiErrorCode := stErrSerialLineControl;
				Out_bolComError := TRUE;
			ELSIF bolErrSend = TRUE THEN
				Out_udiErrorCode := stErrSend;				
				Out_bolComError := TRUE;
			ELSIF bolTimeout = TRUE THEN
				Out_bolProtocolErr := TRUE;
			ELSIF (Out_bolComError = FALSE) AND (Out_bolProtocolErr = FALSE) THEN
				Out_bolComError := TRUE;
			END_IF
			
			// Send NAK to RFID Reader
			IF bolSendNAK = TRUE THEN
				aTxData[0] := cNAK;
				fbSerialSendData(
					pSendData:= ADR(aTxData), 
					Length:= 1, 
					Busy=> bolComSendBusy, 
					Error=> stErrSend, 
					TXbuffer:= stTxBuffer);
					
				IF bolComSendBusy = FALSE THEN
					bolSendNAK := FALSE;
				END_IF
			END_IF
			
			// Acknowledge reset Error bit and informations
			IF (In_bolErrorAck = TRUE) OR (bolIntReset=TRUE) THEN
				intState := cRFD_3964_Wait;
				bolSendNAK := FALSE;
				bolErrSerialLineControl := FALSE; 
				bolErrReceive := FALSE;
				bolErrSend := FALSE;
				bolTimeout := FALSE;
				Out_udiErrorCode := 0;
				Out_bolComError := FALSE;
				Out_bolProtocolErr := FALSE;
				uinCountCall := 0;
				uinCountRetry := 0;
				bolIntReset := FALSE;
				In_bolErrorAck := FALSE;
				bolInitRequest := FALSE;
			END_IF
		
END_CASE

// Write parallel Outputs to commando word
//Out_stEL6outData.Ctrl.2 := bolInitRequest;
//Out_stEL6outData.Ctrl.3 := bolSendContinious;

// make History of States
IF intStateOld <> intState THEN
	udiStateLoop := 9;
	WHILE udiStateLoop > 0 DO
		a_intStateHist[udiStateLoop] := a_intStateHist[udiStateLoop-1];
		udiStateLoop := udiStateLoop-1;
	END_WHILE
	a_intStateHist[0] := intState;
	intStateOld := intState;
	// Time Out control
	// Check timeout
	fbTon(IN:= FALSE, PT:= timQVZ, Q=>bolTimeout );
ELSE
	IF intState <> cRFD_3964_Error THEN
		fbTon(IN:= TRUE, PT:= timQVZ, Q=>bolTimeout );
	END_IF
END_IF

END_FUNCTION_BLOCK

// POUs/Controller/Driver/RFD (RFID Driver)/FB_ExCom
FUNCTION_BLOCK FB_ExCom
VAR_INPUT
	/// Pointer to Received Data Array
	In_pRxData: POINTER TO ARRAY[0..255] OF BYTE;
	/// Pointer to Sending Data Array
	In_pTxData: POINTER TO ARRAY[0..255] OF BYTE;
	/// Amounth of sending data
	In_udiTxCount: UDINT;
	/// Error Acknowledge 
	In_bolErrorAck: BOOL;
END_VAR
VAR_IN_OUT
	/// Command to send Data 1=command; 0=Done
	InOut_bolSend: BOOL;
	/// Command Data received 1=received; 0=Done=Ready for next Data
	InOut_bolRec: BOOL;
END_VAR
VAR_OUTPUT
	/// Amounth of received data
	Out_udiRxCount: UDINT;
	/// Serial interface communication error
	Out_bolComError: BOOL;
	/// Error in protocoll procedure
	Out_bolProtocolErr: BOOL;
	/// Error information to master
	Out_udiErrorCode: UDINT;
END_VAR
VAR
	In_stEL6inData AT %I*: TC2_SERIALCOM.EL6inData22B;
	Out_stEL6outData AT %Q*: TC2_SERIALCOM.EL6outData22B;
	/// Internal Variables
	udiI: UDINT;
	/// Local variable for loops
	udiK: UDINT;
	/// Internal Error Reset
	bolIntReset: BOOL;
	/// Count call trials
	uinCountCall: UINT;
	/// Count call Retrys
	uinCountRetry: UINT;
	/// Temporary value for cecking the sum
	bytCheckValue: BYTE;
	/// Antenna is initializied, until it is not initializied, it send 16#02 in all possible baudrates
	bolSLGInitialized: BOOL := FALSE;
	/// Check Timeout
	bolTimeout: BOOL;
	/// Check Timeout
	bolWait: BOOL;
	/// Send NAK needed
	bolSendNAK: BOOL;
	/// Receive Wait signs
	timWaitReceive: TIME := TIME#5ms;
	/// Receive Wait signs
	timWaitAck: TIME := TIME#400ms;
	/// Sign delay time
	timZVZ: TIME := TIME#45ms;
	/// Time ACK delay
	timQVZ: TIME := TIME#145ms;
	/// Initialisation of the HW card
	bolInitRequest: BOOL;
	/// Setting of the HW Card
	bolSendContinious: BOOL;
	/// Priority at RFID
	bolPriority: BOOL;
	/// Send DLE doubletimes
	bolDLEDouble: BOOL;
	/// New data received
	bolComDataReceived: BOOL;
	/// receiving busy
	bolComRecBusy: BOOL;
	/// Received Data
	udiComSizeReceiveData: UDINT;
	/// Sending busy
	bolComSendBusy: BOOL;
	/// Error at serial line control
	bolErrSerialLineControl: BOOL;
	/// Error at serial line control
	stErrSerialLineControl: ComError_t;
	/// Error at serial line  receiving data
	bolErrReceive: BOOL;
	/// Error at serial line  receiving data
	stErrReceive: ComError_t;
	/// Error at serial line sending data
	bolErrSend: BOOL;
	/// Error at serial line sending data
	stErrSend: ComError_t;
	/// Define Buffer for preparations
	aRxData: ARRAY[0..255] OF BYTE;
	aTxData: ARRAY[0..255] OF BYTE;
	/// Define Buffer for Funciton
	stRxBuffer: TC2_SERIALCOM.ComBuffer;
	/// Transmit data buffer; used with all receive function blocks 
	stTxBuffer: TC2_SERIALCOM.ComBuffer;
	/// Sub Statemachine
	intState: INT := 0;
	intStateOld: INT := 0;
	udiStateLoop: UDINT;
	a_intStateHist: ARRAY[0..9] OF INT;
	udiStateDebug: UDINT;
	udiStateDebugMax: UDINT;
	/// Function for serial communication
	fbSerialLineControl: TC2_SERIALCOM.SerialLineControl;
	fbSerialReceiveData: TC2_SERIALCOM.ReceiveData;
	fbSerialSendData: TC2_SERIALCOM.SendData;
	fbTon: TC2_STANDARD.TON;
	fbWait: TC2_STANDARD.TON;
END_VAR
VAR CONSTANT
	/// Startup
	cExCom_Start: INT := 2500;
	/// Startup
	cExCom_Init: INT := 2501;
	/// Wait for Job
	cExCom_Wait: INT := 2502;
	/// Read recived sign
	cExCom_RxRead: INT := 2504;
	/// Send Data
	cExCom_TxPrepare: INT := 2550;
	/// Send Data
	cExCom_TxSend: INT := 2552;
	/// Error
	cExCom_Error: INT := 2580;
END_VAR

(*__________________________________________________________________________________________________
¦	
¦	Vistaprint Schweiz GmbH
¦	CH - 8401 Winterthur
¦
¦	www.vistaprint.ch - info@vistaprint.ch
¦___________________________________________________________________________________________________

Function desription:
Driver for communication protocoll 3964R
Description in Siemens manual from CP341, A5E02191070-03


History:
Version		Date			Author		Comment
---------------------------------------------------------------------------------------------------
0.00.1		23.07.2013		AVME/PRE	Start history
___________________________________________________________________________________________________*)

// Always
fbSerialLineControl(
	Mode:= TC2_SERIALCOM.ComSerialLineMode_t.SERIALLINEMODE_EL6_22B, 
	pComIn:= ADR(In_stEL6inData), 
	pComOut:= ADR(Out_stEL6outData), 
	SizeComIn:= SIZEOF(In_stEL6inData), 
	Error=> bolErrSerialLineControl, 
	ErrorID=> stErrSerialLineControl, 
	TxBuffer:= stTxBuffer, 
	RxBuffer:= stRxBuffer);
	
// Check timers
IF intState >= cExCom_Wait THEN
	fbWait(PT:= timWaitAck);
END_IF
		
// Startup set correct Step
IF intState < cExCom_Start THEN
	intState := cExCom_Start;
END_IF

// State Machine
CASE intState OF
	cExCom_Start:
		// Clear Buffer
		FOR udiI := 0 TO 255 DO
			aRxData[udiI] := 0;
			aTxData[udiI] := 0;
		END_FOR
		bolSLGInitialized := FALSE;
		
		// Clear counters
		uinCountCall := 0;
		uinCountRetry := 0;
		
		bolInitRequest := FALSE;
		bolSendContinious := FALSE;
		
		
		// Next State
		IF (bolErrSerialLineControl = FALSE) AND (bolTimeout=TRUE) THEN
			intState := cExCom_Init;
		ELSIF (bolErrSerialLineControl = TRUE) THEN
			intState := cExCom_Error;
		END_IF

	// Wait for a job or received Data //	
	cExCom_Init:	
		bolInitRequest := TRUE;
		
		IF (bolErrSerialLineControl = FALSE) AND (bolTimeout=TRUE) THEN	// Initialisation Done
			intState := cExCom_Wait;
		ELSIF (bolErrSerialLineControl = TRUE) THEN
			intState := cExCom_Error;
		END_IF
	
	// Wait for a job or received Data //	
	cExCom_Wait:	
		bolInitRequest := FALSE;
		bolSendNAK := FALSE;
		fbWait.IN := FALSE;
		
		fbSerialReceiveData(
		//	pPrefix:= , // Not used because no prefix in telegram
			LenPrefix:= 0, 
		//	pSuffix:= , // Not used because no suffix in telegram
			LenSuffix:= 0, 
			pReceiveData:= ADR(aRxData), 
			SizeReceiveData:= 255, 
			Timeout:= timWaitReceive, 
		//	Reset:= , 
			DataReceived=> bolComDataReceived, 
			busy=> bolComRecBusy, 
			Error=> stErrReceive, 
			RxTimeout=> bolErrReceive, 
			LenReceiveData=> udiComSizeReceiveData, 
			RXbuffer:= stRxBuffer);
		
		//Check if Data is received
		IF bolComDataReceived = TRUE THEN
			intState := cExCom_RxRead;
		ELSIF (InOut_bolSend = TRUE) AND (bolPriority = FALSE) THEN
			intState := cExCom_TxPrepare;
		END_IF
			
	// Read first signs if new data sending needed //	
	cExCom_RxRead: 
		// Read Signs
		IF (udiComSizeReceiveData >0) THEN
			// Copy Data
			FOR udiI := 0 TO (SIZEOF(aRxData)-1) DO
				In_pRxData^[udiI] := 0;
			END_FOR
			FOR udiI := 0 TO udiComSizeReceiveData-1 DO
				In_pRxData^[udiI] := aRxData[udiI];
			END_FOR
			InOut_bolRec := TRUE;
			Out_udiRxCount := udiComSizeReceiveData;
		END_IF
		
		intState := cExCom_Wait;

		
	// Send Data //		
	cExCom_TxPrepare:
		FOR udiI := 0 TO (SIZEOF(aTxData)-1) DO
			aTxData[udiI] := 0;
		END_FOR
		FOR udiI := 0 TO In_udiTxCount-1 DO
			aTxData[udiI] := In_pTxData^[udiI];
		END_FOR
		intState := cExCom_TxSend;

	cExCom_TxSend:	
		fbSerialSendData(
			pSendData:= ADR(aTxData), 
			Length:= In_udiTxCount, 
			Busy=> bolComSendBusy, 
			Error=> stErrSend, 
			TXbuffer:= stTxBuffer);
			bolSendContinious := TRUE;

			
		// Check transition
		IF (bolComSendBusy = FALSE) AND (stErrSend = 0) THEN
			intState := cExCom_Wait;
			InOut_bolSend := FALSE;
		ELSIF ((bolComSendBusy = TRUE) AND (bolTimeout = TRUE)) OR (stErrSend <> 0) THEN
			bolErrSend := TRUE;
			intState := cExCom_Error;
		END_IF
		

////////////////////////////////////////////////////////////		
		// Error State //
		cExCom_Error:
			IF bolErrSerialLineControl = TRUE THEN
				Out_udiErrorCode := stErrSerialLineControl;
				Out_bolComError := TRUE;
			ELSIF bolErrSend = TRUE THEN
				Out_udiErrorCode := stErrSend;				
				Out_bolComError := TRUE;
			ELSIF bolTimeout = TRUE THEN
				Out_bolProtocolErr := TRUE;
			ELSIF (Out_bolComError = FALSE) AND (Out_bolProtocolErr = FALSE) THEN
				Out_bolComError := TRUE;
			END_IF
		
			
			IF (In_bolErrorAck = TRUE) OR (bolIntReset=TRUE) THEN
				intState := cExCom_Wait;
				bolErrSerialLineControl := FALSE; 
				bolErrReceive := FALSE;
				bolErrSend := FALSE;
				bolTimeout := FALSE;
				Out_udiErrorCode := 0;
				Out_bolComError := FALSE;
				Out_bolProtocolErr := FALSE;
				uinCountCall := 0;
				uinCountRetry := 0;
				In_bolErrorAck := FALSE;
				bolInitRequest := FALSE;
			END_IF
		
END_CASE

// Write parallel Outputs to commando word
//Out_stEL6outData.Ctrl.2 := bolInitRequest;
//Out_stEL6outData.Ctrl.3 := bolSendContinious;

// make History of States
IF intStateOld <> intState THEN
	udiStateLoop := 9;
	WHILE udiStateLoop > 0 DO
		a_intStateHist[udiStateLoop] := a_intStateHist[udiStateLoop-1];
		udiStateLoop := udiStateLoop-1;
	END_WHILE
	a_intStateHist[0] := intState;
	intStateOld := intState;
	// Time Out control
	// Check timeout
	fbTon(IN:= FALSE, PT:= timQVZ, Q=>bolTimeout );
ELSE
	IF intState <> cExCom_Error THEN
		fbTon(IN:= TRUE, PT:= timQVZ, Q=>bolTimeout );
	END_IF
END_IF

END_FUNCTION_BLOCK

// POUs/Controller/Driver/RFD (RFID Driver)/FB_HEXSTRING_TO_ULINT
FUNCTION FB_HEXSTRING_TO_ULINT : ULINT
VAR_INPUT
	in_strSTRING: STRING;
END_VAR
VAR
	uinLenght: UINT;
	intI: INT;
	uliFact: ULINT;
	usiSign: USINT;
	uliReturn: ULINT;
	ausiTemp: ARRAY[0..15] OF USINT;
END_VAR

uinLenght := INT_TO_UINT(TC2_STANDARD.LEN(in_strSTRING));
uliReturn := 0;

IF (uinLenght > 16) THEN
	FB_HEXSTRING_TO_ULINT := 0;
	
ELSE
	MEMCPY(destAddr:=ADR(ausiTemp), srcAddr:=ADR(in_strSTRING), n:=uinLenght);		// COPY to buffer
	intI := UINT_TO_INT(uinLenght)-1;
	uliFact := 1;
	WHILE intI >= 0 DO
		IF (ausiTemp[intI] >= 16#30) AND (ausiTemp[intI] <= 16#39) THEN		// 0=16#30 ...9=16#39
			usiSign := ausiTemp[intI] - 16#30;
		ELSIF (ausiTemp[intI] >= 16#41) AND (ausiTemp[intI] <= 16#46) THEN		// A=16#41 ...F=16#46
			usiSign := ausiTemp[intI] - 55;
		ELSIF (ausiTemp[intI] >= 16#61) AND (ausiTemp[intI] <= 16#66) THEN		// a=16#61 ...f=16#66
			usiSign := ausiTemp[intI] - 87;
		ELSE
			FB_HEXSTRING_TO_ULINT := 0;
			RETURN;
		END_IF
		
		uliReturn := uliReturn + usiSign * uliFact;
		intI := intI - 1;
		uliFact := uliFact * 16;
	END_WHILE
		
END_IF

	FB_HEXSTRING_TO_ULINT := uliReturn;

END_FUNCTION

// POUs/Controller/Driver/RFD (RFID Driver)/FB_RFD
FUNCTION_BLOCK FB_RFD
VAR
	bolActivate: BOOL := TRUE;
	bolInitDone: BOOL;
	bolInitComDone: BOOL;
	///Communication sending is busy to the serial Card
	bolComSend: BOOL;
	/// Size of Sendingdata
	udiComSizeSendData: UDINT;
	///Communication Data Received
	bolComDataReceived: BOOL;
	/// Size of received Data from serial interface
	udiComSizeReceiveData: UDINT;
	///Sdo Setting is busy to the serial Card
	bolSdoBusy: BOOL;
	///Sdo Setting executing
	bolSdoExecute: BOOL;
	/// Antenna Job done
	bolAntennaJobDone: BOOL;
	/// Job Reading is done
	bolReadDone: BOOL;
	/// Job Writing is done
	bolWriteDone: BOOL;
	/// Job Reset SLG is done
	bolResetJobDone: BOOL;
	/// Job Reset SLG has Error
	bolResetJobError: BOOL;
	/// Job Read SLG State is done
	bolSLGJobDone: BOOL;
	/// Job Read SLG State is done
	bolMDSJobDone: BOOL;
	/// Information to SDO Error
	udiSdoErrorNbr: UDINT;
	/// Information to Communication over 3964 protocol Error
	udi3964R_Error_Nbr: UDINT;
	/// Count Reset cycles
	udiResetCount: UDINT;
	/// Count Job Tryals
	udiJobCount: UDINT;
	/// State information from RF ID Tag
	bytRFIDState: BYTE;
	/// driver specific interface
	SIf: T_RFD;
	/// get direct Buffer from Interface
	/// access over mapping!! {attribute 'TcLinkTo':='TIID^Device 1 (EtherCAT)^Box 1 (SGDV-E1 CoE Drive)^2nd Transmit PDO mapping^Status word'}
	aRxData: ARRAY[0..255] OF BYTE;
	aTxData: ARRAY[0..255] OF BYTE;
	/// Function for serial communication
	fbEcCoeSdoWrite: TC2_ETHERCAT.FB_EcCoESdoWrite;
	fbCom_3964R: FB_Com_3964R;
	stStateMachine: T_RFD_StateMachine;
	stSubStateMachine: T_RFD_StateMachine;
	///case variable
	usiCase: USINT;
	///case variable for service cmd's
	usiCaseScmd: USINT;
	/// help values for parameter handling
	sinValue: SINT;
	intValue: INT;
	dinValue: DINT;
	usiValue: USINT;
	uinValue: UINT;
	udiValue: UDINT;
	udiI: UDINT;
	udiLoopBuffer: UDINT;
	udiLoopData: UDINT;
	udiLoopSend: UDINT;
END_VAR

(*__________________________________________________________________________________________________
¦	
¦	Vistaprint Schweiz GmbH
¦	CH - 8401 Winterthur
¦
¦	www.vistaprint.ch - info@vistaprint.ch
¦___________________________________________________________________________________________________

Function desription:
Driver for Simatic RFID Reader and Writer RF310R 6GT2801-1AB10


History:
Version		Date			Author		Comment
---------------------------------------------------------------------------------------------------
0.00.1		09.07.2013		AVME/PRE	Start history
0.00.2		24.09.2013		AVME/KVO	Parameter init from element controller to driver
___________________________________________________________________________________________________*)


IF (bolActivate) THEN // cyclic call enabled
	
	IF (bolInitDone=FALSE) THEN // first cycle -> init
		CtrlInit();
		bolInitDone := TRUE;
	ELSE
		CycleStartDuty();
		
		StateMachine_Service(); // handles asynchron service commands
		
		StateMachine();
		
		CycleEndDuty();
	END_IF
	
END_IF;

METHOD PROTECTED CtrlInit : BOOL
// one time first cyclic call
;
END_METHOD

METHOD PROTECTED CycleEndDuty : BOOL
SIf.strState := THIS^.getCmdState(intCmdState:=stStateMachine.intState,bolState:=TRUE);

IF (stStateMachine.intState<>stStateMachine.intStateNext) THEN
	stStateMachine.intState := stStateMachine.intStateNext;  // set next state for next cycle
END_IF

(***************************************************************
        Function Block Calls
***************************************************************)
END_METHOD

METHOD PROTECTED CycleStartDuty : BOOL
// ----------------------------------------------------------------------------------
// cyclic actions outside of statemachine
fbCom_3964R(
	In_pRxData:= ADR(aRxData), 
	In_pTxData:= ADR(aTxData), 
	In_udiTxCount:= udiComSizeSendData, 
	In_bolErrorAck:= SIf.stErr.bolErrAck, 
	InOut_bolSend:= bolComSend, 
	InOut_bolRec:= bolComDataReceived, 
	Out_udiRxCount=> udiComSizeReceiveData, 
	Out_bolComError=> SIf.stErr.bolComError, 
	Out_bolProtocolErr=> SIf.stErr.bolProtcolError, 
	Out_udiErrorCode=> udi3964R_Error_Nbr);

(* program code at the beginning of each PLC cycle *)
IF bolInitComDone=TRUE THEN
	// Received Data checking and interpreting
	IF bolComDataReceived = TRUE THEN
		CASE aRxData[1] OF
			0:		//16#00 Startup Telegram OR Reset
				IF aRxData[0]= 16#02 THEN 	// Startup Telegram
					IF aRxData[1]= 16#0F THEN
						SIf.stStatus.bolStartupOk := TRUE;				
					END_IF
				ELSE		// Reset Acknowledge
					SIf.stStatus.stSLG_State.worFWVersion := aRxData[3];
					bytRFIDState := aRxData[2];	// Stetebyte copy 1:1
					IF aRxData[2]= 16#00 THEN
						bolResetJobDone := TRUE;
					ELSE
						bolResetJobError := TRUE;
					END_IF
				END_IF
			15:		//16#0F RFID Tag present state
				bytRFIDState := aRxData[2];	// Stetebyte copy 1:1
				IF bytRFIDState=0 THEN
					IF aRxData[4]>0 THEN
						SIf.stStatus.bolPresent := TRUE;
					ELSE
						SIf.stStatus.bolPresent := FALSE;
					END_IF
				END_IF
			1, 65:		//16#01 16#61 Write Acknowledge
				bytRFIDState := aRxData[2];	// Stetebyte copy 1:1
				IF bytRFIDState=0 THEN
					bolWriteDone := TRUE;
				ELSE
					SIf.stErr.bolRFIDError := TRUE;
				END_IF
			2, 66:		//16#02 16#42 Read Acknowledge
				bytRFIDState := aRxData[2];	// Stetebyte copy 1:1
				IF (bytRFIDState=0) AND (SIf.stCur.uinAdressData+SIf.stCur.usiCount <= 255) AND (SIf.stCur.usiCount+6 <= 255) AND (SIf.stCur.usiCount = (aRxData[0]-5)) THEN
					FOR udiLoopBuffer := 0 TO (SIf.stCur.usiCount) DO
						SIf.stCur.pData^[SIf.stCur.uinAdressData+udiLoopBuffer] := aRxData[udiLoopBuffer+6];
					END_FOR	
					bolReadDone := TRUE;
				ELSE
					SIf.stErr.bolRFIDError := TRUE;
				END_IF
			4, 68:		//16#04 16#44 SLG State
				bytRFIDState := aRxData[2];	// Statebyte copy 1:1
				IF bytRFIDState<>0 THEN
					SIf.stErr.bolRFIDError := TRUE;
				ELSE
					IF aRxData[3]=16#01 THEN		// SLG State mode 1
						// HW Type
						SIf.stStatus.stSLG_State.bytHWType := aRxData[4];
						// HW Version
						SIf.stStatus.stSLG_State.worHWVersion := 0;
						SIf.stStatus.stSLG_State.worHWVersion := aRxData[5];
						SIf.stStatus.stSLG_State.worHWVersion := SHL(SIf.stStatus.stSLG_State.worHWVersion,8);
						SIf.stStatus.stSLG_State.worHWVersion := SIf.stStatus.stSLG_State.worHWVersion OR aRxData[6];
						// URL Version
						SIf.stStatus.stSLG_State.worURLVersion := 0;
						SIf.stStatus.stSLG_State.worURLVersion := aRxData[7];
						SIf.stStatus.stSLG_State.worURLVersion := SHL(SIf.stStatus.stSLG_State.worURLVersion,8);
						SIf.stStatus.stSLG_State.worURLVersion := SIf.stStatus.stSLG_State.worURLVersion OR aRxData[8];
						// FW Type
						SIf.stStatus.stSLG_State.bytFWType := aRxData[9];
						// FW Version
						SIf.stStatus.stSLG_State.worFWVersion := 0;
						SIf.stStatus.stSLG_State.worFWVersion := aRxData[10];
						SIf.stStatus.stSLG_State.worFWVersion := SHL(SIf.stStatus.stSLG_State.worFWVersion,8);
						SIf.stStatus.stSLG_State.worFWVersion := SIf.stStatus.stSLG_State.worFWVersion OR aRxData[11];
						// TR Type
						SIf.stStatus.stSLG_State.bytDriverType := aRxData[12];
						// TR Version
						SIf.stStatus.stSLG_State.worDriverVersion := 0;
						SIf.stStatus.stSLG_State.worDriverVersion := aRxData[13];
						SIf.stStatus.stSLG_State.worDriverVersion := SHL(SIf.stStatus.stSLG_State.worDriverVersion,8);
						SIf.stStatus.stSLG_State.worDriverVersion := SIf.stStatus.stSLG_State.worDriverVersion OR aRxData[14];
						// Serial Interface
						SIf.stStatus.stSLG_State.bytComm := aRxData[15];
						// Serial Interface Baud Rate
						SIf.stStatus.stSLG_State.bytBaud := aRxData[16];
						// sending power (only RF380R)
						SIf.stStatus.stSLG_State.bytPower := aRxData[20];
						// Number of maximal tags in the field
						SIf.stStatus.stSLG_State.bytMtag := aRxData[21];
						// air interface 0=RF300; 1=ISO generall; 3=ISO infineon Chip; 4=ISO Fujitsu; 5=ISO NXP; 6=ISO TI; 7=ISO ST
						SIf.stStatus.stSLG_State.bytFtim := aRxData[23];
						// State antenna 1=ON; 2=OFF
						SIf.stStatus.stSLG_State.bytAntenna := aRxData[25];
						// Tag presence 0=No presence; 1=prexence
						SIf.stStatus.stSLG_State.bytPresence := aRxData[27];
					ELSE		// SLG Diagnose Mode 6
						// Errorcounter inactive mode
						SIf.stStatus.stSLG_Diag.usiFZP := aRxData[4];
						// Counter abort
						SIf.stStatus.stSLG_Diag.usiABZ := aRxData[5];
						// Errorcounter code errors
						SIf.stStatus.stSLG_Diag.usiCFZ := aRxData[6];
						// Errorcounter signature errors
						SIf.stStatus.stSLG_Diag.usiSFZ := aRxData[7];
						// Errorcounter CRC
						SIf.stStatus.stSLG_Diag.usiCRCFZ := aRxData[8];
						// Actual command state
						SIf.stStatus.stSLG_Diag.usiBSTAT := aRxData[9];
						// Counter interface errors to host (Parity, BCC, Frame)
						SIf.stStatus.stSLG_Diag.usiASMFZ := aRxData[10];
					END_IF
				END_IF
				bolSLGJobDone := TRUE;

			11, 75:		//16#0B 16#4B MDS State
				bytRFIDState := aRxData[2];	// Statebyte copy 1:1
				IF bytRFIDState<>0 THEN
					SIf.stErr.bolRFIDError := TRUE;
				ELSE
					// UID
					SIf.stStatus.abyteUID[7] := aRxData[4];
					SIf.stStatus.abyteUID[6] := aRxData[5];
					SIf.stStatus.abyteUID[5] := aRxData[6];
					SIf.stStatus.abyteUID[4] := aRxData[7];
					SIf.stStatus.abyteUID[3] := aRxData[8];
					SIf.stStatus.abyteUID[2] := aRxData[9];
					SIf.stStatus.abyteUID[1] := aRxData[10];
					SIf.stStatus.abyteUID[0] := aRxData[11];
						
					IF aRxData[3]=16#01 THEN		// MDS State mode 1 RF300
						SIf.stStatus.stMDS_State.bytMDSType := aRxData[12];
						SIf.stStatus.stMDS_State.bytLockState := aRxData[13];
						SIf.stStatus.stMDS_State.worMemSize := 0;		// No information at this type			
						SIf.stStatus.stMDS_State.bytLockState := 0;		// No information at this type
						SIf.stStatus.stMDS_State.bytBlockSize := 0;		// No information at this type
						SIf.stStatus.stMDS_State.bytBlockNo := 0;		// No information at this type
					ELSIF aRxData[3]=16#02 THEN		// MDS Diagnose mode 2 RF300
						SIf.stStatus.stMDS_Diag.usiLFD := aRxData[12];
						SIf.stStatus.stMDS_Diag.usiFZP := aRxData[13];
						SIf.stStatus.stMDS_Diag.usiFZA := aRxData[14];
						SIf.stStatus.stMDS_Diag.usiANWZ := aRxData[15];
					ELSIF aRxData[3]=16#03 THEN		// MDS State mode 3 ISO
						SIf.stStatus.stMDS_State.bytMDSType := aRxData[12];
						SIf.stStatus.stMDS_State.bytVersion := aRxData[13];
						SIf.stStatus.stMDS_State.worMemSize := aRxData[14]*256 + aRxData[15];				
						SIf.stStatus.stMDS_State.bytLockState := aRxData[16];
						SIf.stStatus.stMDS_State.bytBlockSize := aRxData[17];
						SIf.stStatus.stMDS_State.bytBlockNo := aRxData[18];
					END_IF
				END_IF
				bolMDSJobDone := TRUE;
		
					
			10, 42:		//16#2A SET Antenna
				bytRFIDState := aRxData[2];	// Stetebyte copy 1:1
				IF bytRFIDState=0 THEN
					bolAntennaJobDone := TRUE;
				ELSE
					SIf.stErr.bolRFIDError := TRUE;
				END_IF
			16#FF:		//Communication Check to SLG
				SIf.stStatus.bolL_UEB := TRUE;		
		
		END_CASE
	// Data processed, reset bol to ACK
	bolComDataReceived := FALSE;
	END_IF
END_IF

// always go to Error 
(*KVO no auto start because config write from RFW-slow programm
IF (stStateMachine.intState<cRFD_STA_PowerOnBusy) AND (stStateMachine.intState<>cRFD_STA_Error) THEN
	stStateMachine.intStateNext := cRFD_STA_PowerOnBusy;
ELS*)
IF (SIf.stErr.bolErrorActive) AND 
	(stStateMachine.intState<>cRFD_STA_Error)  THEN
	stStateMachine.intStateNext := cRFD_STA_Error;
// always go to PowerOff 
ELSIF ((SIf.intCmd=cRFD_CMD_CTRL_OFF)) AND 
	(stStateMachine.intState<>cRFD_STA_Off) AND 
	(stStateMachine.intState<>cRFD_STA_Error) THEN
	stStateMachine.intStateNext := cRFD_STA_Off;
ELSIF ((SIf.intCmd=RFD_Cmd.cRFD_CMD_CTRL_ON) AND (stStateMachine.intState<>cRFD_STA_PowerOnBusy)) THEN
	stStateMachine.intStateNext := cRFD_STA_PowerOnBusy;
END_IF

SIf.strCmd := THIS^.getCmdState(intCmdState:=SIf.intCmd,bolState:=FALSE);
END_METHOD

METHOD FB_init : BOOL
VAR_INPUT
	///if TRUE, the retain variables are initialized (warm start / cold start)
	bInitRetains: BOOL;
	///if TRUE, the instance afterwards gets moved into the copy code (online change)
	bInCopyCode: BOOL;
END_VAR
VAR
	udiTaskCnt: UDINT;
	ii: UINT;
END_VAR
SIf.intCmd := cRFD_CMD_DONE;
SIf.intServiceCmd := cRFD_CMD_DONE; // not used at the moment
stStateMachine.intStateLastCycle  := cRFD_CMD_DONE; //EntryStop of power BASE_PLC.OFF enable

// Vaild Values into the Configuration
SIf.stCfg.usiFtimSetting := E_Typ_Ftim.RF300;

// Communication Settings
SIf.stCfg.eTyp := E_Typ_RFW.RF310R;
SIf.stCfg.uinBaudrate := UINT_TO_USINT(E_Typ_Baudrate.baud_57600);
SIf.stCfg.stNetId := '192.168.70.26.3.1';
SIf.stCfg.uinSlaveAddr := 1002;
END_METHOD

METHOD PROTECTED getCmdState : STRING
VAR_INPUT
	intCmdState: INT;
	bolState: BOOL;
END_VAR
// get string cmd/state string information in runtime
IF (bolState=FALSE) THEN
	// cmd's
	CASE intCmdState OF
		cRFD_CMD_DONE: 
			getCmdState := 'cRFD_CMD_DONE';
		cRFD_CMD_CTRL_ON: 
			getCmdState := 'cRFD_CMD_CTRL_ON';
		cRFD_CMD_CTRL_OFF: 
			getCmdState := 'cRFD_CMD_CTRL_OFF';
		cRFD_CMD_Write: 
			getCmdState := 'cRFD_CMD_Write';
		cRFD_CMD_Read: 
			getCmdState := 'cRFD_CMD_Read';
		cRFD_CMD_MDS: 
			getCmdState := 'cRFD_CMD_MDS';
		cRFD_CMD_SLG: 
			getCmdState := 'cRFD_CMD_SLG';
	END_CASE;
ELSE

// States
	CASE intCmdState OF
		cRFD_STA_Error: 
			getCmdState := 'cRFD_STA_Error';
		cRFD_STA_WaitForJob: 
			getCmdState := 'cRFD_STA_WaitForJob';
		cRFD_STA_PowerOnBusy: 
			getCmdState := 'cRFD_STA_PowerOnBusy';
		cRFD_STA_OffBusy: 
			getCmdState := 'cRFD_STA_OffBusy';
		cRFD_STA_Off: 
			getCmdState := 'cRFD_STA_Off';
		cRFD_STA_WriteBusy: 
			getCmdState := 'cRFD_STA_WriteBusy';
		cRFD_STA_ReadBusy: 
			getCmdState := 'cRFD_STA_ReadBusy';
		cRFD_STA_TagInitBusy: 
			getCmdState := 'cRFD_STA_TagInitBusy';
		cRFD_STA_CheckBusy: 
			getCmdState := 'cRFD_STA_CheckBusy';
		cRFD_STA_MDSBusy: 
			getCmdState := 'cRFD_STA_MDSBusy';
		cRFD_STA_SLGBusy: 
			getCmdState := 'cRFD_STA_SLGBusy';

	END_CASE;
END_IF
END_METHOD

METHOD getSIf : POINTER TO T_RFD
getSIf := ADR(SIf);
END_METHOD

METHOD PROTECTED sta_CheckBusy : BOOL
// state implemetation
//--------------------------------------------------------------------------------------
// Entry action
	IF (stStateMachine.intState<>stStateMachine.intStateLastCycle) THEN
		stStateMachine.intStateLastCycle := stStateMachine.intState;
			// Byte 0 => Lenght
			aTxData[0] := 2;
			// Byte 1 => Command read 4=single; 14=continious
			aTxData[1] := 16#FF;
			// Byte 2 => Spare
			aTxData[2] := 0;
						
			udiComSizeSendData := 3;
			bolComSend := TRUE;	
			SIf.stStatus.bolL_UEB := FALSE;
	END_IF


//--------------------------------------------------------------------------------------
// Cyclic action
	IF (stStateMachine.intState=stStateMachine.intStateLastCycle) THEN

		
		// State Change Condition
		IF (SIf.stErr.bolErrorActive = TRUE) THEN
			stStateMachine.intStateNext := cRFD_STA_Error;
		ELSIF (SIf.stStatus.bolL_UEB = TRUE) THEN
			stStateMachine.intStateNext := cRFD_STA_WaitForJob;
		END_IF
		
	END_IF

//--------------------------------------------------------------------------------------
// Exit action
	IF (stStateMachine.intState<>stStateMachine.intStateNext) THEN
		SIf.intCmd := cRFD_CMD_DONE;
	END_IF
END_METHOD

METHOD PROTECTED sta_Error : BOOL
// state implemetation
//--------------------------------------------------------------------------------------
// Entry action
	IF (stStateMachine.intState<>stStateMachine.intStateLastCycle) THEN
		stStateMachine.intStateHistory := stStateMachine.intStateLastCycle;
		stStateMachine.intStateLastCycle := stStateMachine.intState;
		
	END_IF


//--------------------------------------------------------------------------------------
// Cyclic action
	IF (stStateMachine.intState=stStateMachine.intStateLastCycle) THEN
		SIf.stErr.bolErrorActive := TRUE;
		IF (SIf.stErr.bolComError = TRUE) OR (SIf.stErr.bolProtcolError = TRUE) THEN
			SIf.stErr.udiErrorID := udi3964R_Error_Nbr;
		ELSIF SIf.stErr.bolSDOError = TRUE THEN
			SIf.stErr.udiErrorID := udiSdoErrorNbr;
		ELSIF (udiResetCount >=SIf.stCfg.udiRetry) OR (udiJobCount >= SIf.stCfg.udiRetry) THEN
			SIf.stErr.udiErrorID := SIf.stCfg.udiRetry;
		ELSE
			SIf.stErr.udiErrorID := 0;
		END_IF

		
		// State Change Condition
		IF (SIf.stErr.bolErrAck = TRUE) THEN
			// Reset all active errors
			SIf.stErr.bolErrorActive := FALSE;
			SIf.stErr.bolComError := FALSE;
			SIf.stErr.bolProtcolError := FALSE;
			SIf.stErr.bolSDOError := FALSE;
			SIf.stErr.udiErrorID := 0;
		
		
			IF stStateMachine.intStateHistory < cRFD_STA_WaitForJob THEN
				stStateMachine.intStateNext := cRFD_STA_Off;
			ELSE
				stStateMachine.intStateNext := cRFD_STA_WaitForJob;		
			END_IF
		END_IF
	END_IF




//--------------------------------------------------------------------------------------
// Exit action
	IF (stStateMachine.intState<>stStateMachine.intStateNext) THEN
		;
	END_IF
END_METHOD

METHOD PROTECTED sta_MDSBusy : BOOL
// state implemetation
//--------------------------------------------------------------------------------------
// Entry action
	IF (stStateMachine.intState<>stStateMachine.intStateLastCycle) THEN
		stStateMachine.intStateLastCycle := stStateMachine.intState;
			stSubStateMachine.intState := cRFD_SUB_Write1;
			stSubStateMachine.intStateNext := cRFD_SUB_Write1;
	END_IF


//--------------------------------------------------------------------------------------
// Cyclic action
	IF (stStateMachine.intState=stStateMachine.intStateLastCycle) THEN
		CASE stSubStateMachine.intState OF
			cRFD_SUB_Write1:
				// Byte 0 => Lenght
				aTxData[0] := 5;
				// Byte 1 => Command read 4=single; 14=continious
				aTxData[1] := 16#B;
				// Byte 2 => Spare
				aTxData[2] := 0;
				// Byte 3 => Mode
				aTxData[3] := 3;
				// Byte 4 => Spare
				aTxData[4] := 0;
				// Byte 5 => Spare
				aTxData[5] := 0; 

						
				udiComSizeSendData := 6;
				bolComSend := TRUE;	
				stSubStateMachine.intState := cRFD_SUB_Wait1;
		
			cRFD_SUB_Wait1:
				IF bolMDSJobDone = TRUE THEN
					stSubStateMachine.intState := cRFD_SUB_SubStatesEnd;
					bolMDSJobDone := FALSE;
				END_IF
		cRFD_SUB_SubStatesEnd:
				;
				
		END_CASE
		
		// State Change Condition
		IF (SIf.stErr.bolComError = TRUE) OR ((SIf.stErr.bolRFIDError = TRUE) AND (udiJobCount > SIf.stCfg.udiRetry)) THEN
			stStateMachine.intStateNext := cRFD_STA_Error;
		ELSIF (SIf.stErr.bolRFIDError = TRUE) THEN
			udiJobCount := udiJobCount + 1;
			stStateMachine.intStateLastCycle := 0; // Startcycle again
		ELSIF (stSubStateMachine.intState = cRFD_SUB_SubStatesEnd) THEN
			udiJobCount := 0;
			stStateMachine.intStateNext := cRFD_STA_WaitForJob;
		END_IF
		
	END_IF

//--------------------------------------------------------------------------------------
// Exit action
	IF (stStateMachine.intState<>stStateMachine.intStateNext) THEN
		SIf.intCmd := cRFD_CMD_DONE;
	END_IF
END_METHOD

METHOD PROTECTED sta_Off : BOOL
// state implemetation
//--------------------------------------------------------------------------------------
// Entry action
	IF (stStateMachine.intState<>stStateMachine.intStateLastCycle) THEN
		stStateMachine.intStateLastCycle := stStateMachine.intState;
		
	END_IF


//--------------------------------------------------------------------------------------
// Cyclic action
	IF (stStateMachine.intState=stStateMachine.intStateLastCycle) THEN

		
		// State Change Condition
		IF (FALSE) THEN
			stStateMachine.intStateNext := cRFD_STA_Error;
		ELSIF (SIf.intCmd=cRFD_CMD_CTRL_ON) THEN
			stStateMachine.intStateNext := cRFD_STA_PowerOnBusy;
		END_IF
		
	END_IF

//--------------------------------------------------------------------------------------
// Exit action
	IF (stStateMachine.intState<>stStateMachine.intStateNext) THEN
		;
	END_IF
END_METHOD

METHOD PROTECTED sta_OffBusy : BOOL
// state implemetation
//--------------------------------------------------------------------------------------
// Entry action
	IF (stStateMachine.intState<>stStateMachine.intStateLastCycle) THEN
		stStateMachine.intStateLastCycle := stStateMachine.intState;
			IF SIf.stStatus.bolOn = TRUE THEN
				stSubStateMachine.intState := cRFD_SUB_Prepare;		// First Time set Baudrate and communication Settings
				stSubStateMachine.intStateNext := cRFD_SUB_Prepare;		// First Time set Baudrate and communication Settings
			ELSE
				stSubStateMachine.intState := cRFD_SUB_SubStatesEnd;
				stSubStateMachine.intStateNext := cRFD_SUB_SubStatesEnd;
			END_IF
			bolAntennaJobDone := FALSE;
	END_IF


//--------------------------------------------------------------------------------------
// Cyclic action
	IF (stStateMachine.intState=stStateMachine.intStateLastCycle) THEN
		
		// main statemachine of base controller
		CASE stSubStateMachine.intState OF
			cRFD_SUB_Prepare: 
				FOR udiI := 0 TO SIZEOF(aTxData) DO
					aTxData[udiI] := 0;
				END_FOR
				
				/// Send Command to set antenna OFF
				// Byte 0 => Lenght of telegram
				aTxData[0] := 3;
				// Byte 1 => Command Antenna job
				aTxData[1] := 16#A;
				// Byte 2 => Spare
				aTxData[2] := 0;
				// Byte 3 => Mode 1=On; 2=Off
				aTxData[3] := 2;
				
				udiComSizeSendData := 4;
				bolComSend := TRUE;
				stSubStateMachine.intStateNext := cRFD_SUB_SendBusy;
		
		cRFD_SUB_SendBusy:		
				IF ((SIf.stErr.bolComError = FALSE) AND (bolComSend = FALSE)) THEN
					stSubStateMachine.intStateNext := cRFD_SUB_WaitAnswer;
				END_IF

			cRFD_SUB_WaitAnswer:
				IF (bolAntennaJobDone = TRUE) THEN
					SIf.stStatus.bolOn := FALSE;
					stSubStateMachine.intStateNext := cRFD_SUB_SubStatesEnd;
				END_IF
				
			cRFD_SUB_SubStatesEnd:
				;
		END_CASE
		
		stSubStateMachine.intStateLastCycle := stSubStateMachine.intState;
		IF (stSubStateMachine.intState<>stSubStateMachine.intStateNext) THEN
			stSubStateMachine.intState := stSubStateMachine.intStateNext;  // set next state for next cycle
		END_IF
		

		// State Change Condition
		IF (stSubStateMachine.intStateNext = cRFD_SUB_SubStatesEnd) THEN
			stStateMachine.intStateNext := cRFD_STA_Off;
		END_IF
		
	END_IF


//--------------------------------------------------------------------------------------
// Exit action
	IF (stStateMachine.intState<>stStateMachine.intStateNext) THEN
		SIf.intCmd := cRFD_CMD_DONE;
		SIf.stStatus.bolOn := FALSE;
	END_IF
END_METHOD

METHOD PROTECTED sta_PowerOnBusy : BOOL
// state implemetation
//--------------------------------------------------------------------------------------
// Entry action
	IF (stStateMachine.intState<>stStateMachine.intStateLastCycle) THEN
		stStateMachine.intStateLastCycle := stStateMachine.intState;

			//IF bolInitComDone=FALSE THEN
				// direct write parameter doesn't work!! KVO 17.09.2013 with new Kannegiesser RFID
				// Feedback rx[0..2] 255 4 251 -> Baudrate/task time not 2ms
				// no Feedback -> parameter set? estimated  rx[0..2] 1 0 1
				// decision with Rolf Engelputzeder 18.09.2013 
				// don't use write parameter at the moment:
				stSubStateMachine.intState := cRFD_SUB_SubStatesEnd;// cRFD_SUB_ClearBuffer;		// First Time set Baudrate and communication Settings
				stSubStateMachine.intStateNext := cRFD_SUB_SubStatesEnd;// cRFD_SUB_ClearBuffer;		// First Time set Baudrate and communication Settings
				bolInitComDone := TRUE; // old without this condition
				
				(*
				// original set parameter to RFID
				IF bolInitComDone=FALSE THEN
					stSubStateMachine.intState := cRFD_SUB_SetBaudrate;		// First Time set Baudrate and communication Settings
					stSubStateMachine.intStateNext := cRFD_SUB_SetBaudrate;		// First Time set Baudrate and communication Settings
				ELSE
					stSubStateMachine.intState := cRFD_SUB_ClearBuffer;
					stSubStateMachine.intStateNext := cRFD_SUB_ClearBuffer;
				END_IF
				*)
			//END_IF
			
			bolSdoExecute := FALSE;
			bolResetJobDone := FALSE;
	END_IF


//--------------------------------------------------------------------------------------
// Cyclic action
	IF (stStateMachine.intState=stStateMachine.intStateLastCycle) THEN
		
		// main statemachine of base controller
		CASE stSubStateMachine.intState OF
			cRFD_SUB_SetBaudrate:
				IF stSubStateMachine.intStateLastCycle <> stSubStateMachine.intState THEN
					stSubStateMachine.intStateLastCycle := stSubStateMachine.intState;
				END_IF
				fbEcCoeSdoWrite(
					sNetId:= SIf.stCfg.stNetId, 
					nSlaveAddr:= SIf.stCfg.uinSlaveAddr, 
					nIndex:= SIf.stCfg.uinCoeIndexComSettings, 
					nSubIndex:= SIf.stCfg.usiCoeSubindexComBaudrate, 
					pSrcBuf:= ADR(SIf.stCfg.uinBaudrate), 
					cbBufLen:= SIZEOF(SIf.stCfg.uinBaudrate), 
					bExecute:= bolSdoExecute, 
					tTimeout:= DEFAULT_ADS_TIMEOUT, 
					bBusy=> bolSdoBusy, 
					bError=> SIf.stErr.bolSDOError, 
					nErrId=> udiSdoErrorNbr);
					
					
				IF 	(bolSdoExecute = TRUE) THEN
					IF ((SIf.stErr.bolSDOError = FALSE) AND (bolSdoBusy = FALSE)) THEN
						bolSdoExecute := FALSE;
						stSubStateMachine.intStateNext := cRFD_SUB_ClearBuffer;
					END_IF
				ELSE
					bolSdoExecute := TRUE;
				END_IF
				
			
			cRFD_SUB_SetComSettings:
				IF stSubStateMachine.intStateLastCycle <> stSubStateMachine.intState THEN
					stSubStateMachine.intStateLastCycle := stSubStateMachine.intState;
				END_IF
				fbEcCoeSdoWrite(
					sNetId:= SIf.stCfg.stNetId, 
					nSlaveAddr:= SIf.stCfg.uinSlaveAddr, 
					nSubIndex:= SIf.stCfg.usiCoeSubindexComDataframe, 
					nIndex:= SIf.stCfg.uinCoeIndexComSettings, 
					pSrcBuf:= ADR(SIf.stCfg.uinComSettings), 
					cbBufLen:= SIZEOF(SIf.stCfg.uinComSettings), 
					bExecute:= bolSdoExecute, 
					tTimeout:= T#2S, 
					bBusy=> bolSdoBusy, 
					bError=> SIf.stErr.bolSDOError, 
					nErrId=> udiSdoErrorNbr);
					
				IF 	(bolSdoExecute = TRUE) THEN
					IF ((SIf.stErr.bolSDOError = FALSE) AND (bolSdoBusy = FALSE)) THEN
						bolSdoExecute := FALSE;
						stSubStateMachine.intStateNext := cRFD_SUB_ClearBuffer;
					END_IF
				ELSE
					bolSdoExecute := TRUE;
				END_IF

	
			cRFD_SUB_ClearBuffer: 	 
				IF stSubStateMachine.intStateLastCycle <> stSubStateMachine.intState THEN
					stSubStateMachine.intStateLastCycle := stSubStateMachine.intState;
				END_IF
				bolInitComDone := TRUE;
				IF (SIf.stErr.bolComError = FALSE) THEN
					stSubStateMachine.intStateNext := cRFD_SUB_InitString;
				END_IF

				
			cRFD_SUB_InitString: 
				IF stSubStateMachine.intStateLastCycle <> stSubStateMachine.intState THEN
					stSubStateMachine.intStateLastCycle := stSubStateMachine.intState;
					aTxData[0] := 10;
					// Byte 1 => Spare
					aTxData[1] := 0;
					// Byte 2 => Spare
					aTxData[2] := 0;
					// Byte 3 => Spare
					aTxData[3] := 0;
					// Byte 4 => Reset Parameter
					aTxData[4] := 16#25; // SIf.stCfg.usiResetParameter;
					// Byte 5 => Reset option
					aTxData[5] := 16#2; //SIf.stCfg.usiResetOption1;
					// Byte 6 => dili = Setting of sendepower antenna (only RF380R)
					aTxData[6] := 0; //0;
					// Byte 7 => Spare
					aTxData[7] := 0;
					// Byte 8 => mtag = Maximal value of tags in field
					aTxData[8] := 1;
					// Byte 9 => Spare
					aTxData[9] := 0;
					// Byte 10 => ftim = Setting for the Air interface
					aTxData[10] := 1;
					
					udiComSizeSendData := 11;
					bolComSend := TRUE;
				END_IF
			
				IF ((SIf.stErr.bolComError = 0) AND (bolComSend = FALSE)) THEN	 //AND (bolComSendBusy_old = TRUE)
					stSubStateMachine.intStateNext := cRFD_SUB_CheckPon;
				END_IF

			cRFD_SUB_CheckPon:
				IF (bolResetJobDone = TRUE) THEN
					stSubStateMachine.intStateNext := cRFD_SUB_SubStatesEnd;
				ELSIF (bolResetJobError =TRUE) AND (udiResetCount < SIf.stCfg.udiRetry) THEN
					bolResetJobError := FALSE;
					udiResetCount := udiResetCount + 1;
					stSubStateMachine.intStateNext := cRFD_SUB_InitString;
				END_IF
				
			cRFD_SUB_SubStatesEnd:
				;
		END_CASE
		
		stSubStateMachine.intStateLastCycle := stSubStateMachine.intState;
		IF (stSubStateMachine.intState<>stSubStateMachine.intStateNext) THEN
			stSubStateMachine.intState := stSubStateMachine.intStateNext;  // set next state for next cycle
			//stSubStateMachine.udiTimeInState_ms := 0; // reset timer
			// log state change -> open point
		//ELSE
			// increment time in state	
			//stSubStateMachine.intStateLastCycle := stSubStateMachine.udiTimeInState_ms + me.FUBInfo.udiSample_ms;
		END_IF
		

		// State Change Condition
		IF (SIf.stErr.bolComError = TRUE) OR (SIf.stErr.bolSDOError = TRUE) OR (udiResetCount >= SIf.stCfg.udiRetry) THEN
			stStateMachine.intStateNext := cRFD_STA_Error;
		ELSIF (stSubStateMachine.intStateNext = cRFD_SUB_SubStatesEnd) THEN
			stStateMachine.intStateNext := cRFD_STA_WaitForJob;
		END_IF
		
	END_IF


//--------------------------------------------------------------------------------------
// Exit action
	IF (stStateMachine.intState<>stStateMachine.intStateNext) THEN
		SIf.intCmd := cRFD_CMD_DONE;
		SIf.stStatus.bolStartupOk := TRUE;
		SIf.stStatus.bolInitOk := TRUE;
		SIf.stStatus.bolOn := TRUE;
	END_IF
END_METHOD

METHOD PROTECTED sta_ReadBusy : BOOL
// state implemetation
//--------------------------------------------------------------------------------------
// Entry action
	IF (stStateMachine.intState<>stStateMachine.intStateLastCycle) THEN
		stStateMachine.intStateLastCycle := stStateMachine.intState;
			// Byte 0 => Lenght
			aTxData[0] := 5;
			// Byte 1 => Command read 2=single; 12=continious
			aTxData[1] := 2;
			// Byte 2 => Spare
			aTxData[2] := 0;
			// Byte 3 => Adress MSB
			uinValue := SIf.stCur.uinAdressTag;
			uinValue := ROL(uinValue,8);
			aTxData[3] := UINT_TO_USINT(uinValue);
			// Byte 4 => Adress LSB
			aTxData[4] := UINT_TO_USINT(SIf.stCur.uinAdressTag);
			// Byte 5 =>Lenght
			aTxData[5] := SIf.stCur.usiCount; 
					
			udiComSizeSendData := 6;
			bolComSend := TRUE;	
	END_IF


//--------------------------------------------------------------------------------------
// Cyclic action
	IF (stStateMachine.intState=stStateMachine.intStateLastCycle) THEN


		
		// State Change Condition
		IF (SIf.stErr.bolComError = TRUE) OR ((SIf.stErr.bolRFIDError = TRUE) AND (udiJobCount > SIf.stCfg.udiRetry)) THEN
			stStateMachine.intStateNext := cRFD_STA_Error;
		ELSIF (SIf.stErr.bolRFIDError = TRUE) THEN
			udiJobCount := udiJobCount + 1;
			stStateMachine.intStateLastCycle := 0; // Startcycle again
		ELSIF ((SIf.stErr.bolComError = 0) AND (bolReadDone = TRUE)) THEN
			bolReadDone := FALSE;
			udiJobCount := 0;
			stStateMachine.intStateNext := cRFD_STA_WaitForJob;
		END_IF
		
	END_IF

//--------------------------------------------------------------------------------------
// Exit action
	IF (stStateMachine.intState<>stStateMachine.intStateNext) THEN
		SIf.intCmd := cRFD_CMD_DONE;
	END_IF
END_METHOD

METHOD PROTECTED sta_SLGBusy : BOOL
// state implemetation
//--------------------------------------------------------------------------------------
// Entry action
	IF (stStateMachine.intState<>stStateMachine.intStateLastCycle) THEN
		stStateMachine.intStateLastCycle := stStateMachine.intState;
			stSubStateMachine.intState := cRFD_SUB_Write1;
			stSubStateMachine.intStateNext := cRFD_SUB_Write1;
	END_IF


//--------------------------------------------------------------------------------------
// Cyclic action
	IF (stStateMachine.intState=stStateMachine.intStateLastCycle) THEN
		CASE stSubStateMachine.intState OF
			cRFD_SUB_Write1:
				// Byte 0 => Lenght
				aTxData[0] := 6;
				// Byte 1 => Command read 4=single; 14=continious
				aTxData[1] := 4;
				// Byte 2 => Spare
				aTxData[2] := 0;
				// Byte 3 => Mode
				aTxData[3] := 1;
				// Byte 4 => Spare
				aTxData[4] := 0;
				// Byte 5 => Spare
				aTxData[5] := 0; 
				// Byte 6 => Spare
				aTxData[6] := 0; 
						
				udiComSizeSendData := 7;
				bolComSend := TRUE;	
				stSubStateMachine.intState := cRFD_SUB_Wait1;
		
			cRFD_SUB_Wait1:
				IF bolSLGJobDone = TRUE THEN
					stSubStateMachine.intState := cRFD_SUB_Write6;
					bolSLGJobDone := FALSE;
				END_IF
			cRFD_SUB_Write6:
				// Byte 0 => Lenght
				aTxData[0] := 6;
				// Byte 1 => Command read 4=single; 14=continious
				aTxData[1] := 4;
				// Byte 2 => Spare
				aTxData[2] := 0;
				// Byte 3 => Mode
				aTxData[3] := 6;
				// Byte 4 => Spare
				aTxData[4] := 0;
				// Byte 5 => Spare
				aTxData[5] := 0; 
				// Byte 6 => Spare
				aTxData[6] := 0; 
						
				udiComSizeSendData := 7;
				bolComSend := TRUE;	
				stSubStateMachine.intState := cRFD_SUB_Wait6;
		
			cRFD_SUB_Wait6:
				IF bolSLGJobDone = TRUE THEN
					stSubStateMachine.intState := cRFD_SUB_SubStatesEnd;
					bolSLGJobDone := FALSE;
				END_IF
			
			cRFD_SUB_SubStatesEnd:
				;
				
		END_CASE
		
		// State Change Condition
		IF (SIf.stErr.bolComError = TRUE) OR ((SIf.stErr.bolRFIDError = TRUE) AND (udiJobCount > SIf.stCfg.udiRetry)) THEN
			stStateMachine.intStateNext := cRFD_STA_Error;
		ELSIF (SIf.stErr.bolRFIDError = TRUE) THEN
			udiJobCount := udiJobCount + 1;
			stStateMachine.intStateLastCycle := 0; // Startcycle again
		ELSIF (stSubStateMachine.intState = cRFD_SUB_SubStatesEnd) THEN
			udiJobCount := 0;
			stStateMachine.intStateNext := cRFD_STA_WaitForJob;
		END_IF
		
	END_IF

//--------------------------------------------------------------------------------------
// Exit action
	IF (stStateMachine.intState<>stStateMachine.intStateNext) THEN
		SIf.intCmd := cRFD_CMD_DONE;
	END_IF
END_METHOD

METHOD PROTECTED sta_TagInitBusy : BOOL
// state implemetation
//--------------------------------------------------------------------------------------
// Entry action
	IF (stStateMachine.intState<>stStateMachine.intStateLastCycle) THEN
		stStateMachine.intStateLastCycle := stStateMachine.intState;
		
	END_IF


//--------------------------------------------------------------------------------------
// Cyclic action
	IF (stStateMachine.intState=stStateMachine.intStateLastCycle) THEN

		
		// State Change Condition
		IF (FALSE) THEN
			stStateMachine.intStateNext := cRFD_STA_Error;
		ELSIF (TRUE) THEN
			stStateMachine.intStateNext := cRFD_STA_WaitForJob;
		END_IF
		
	END_IF

//--------------------------------------------------------------------------------------
// Exit action
	IF (stStateMachine.intState<>stStateMachine.intStateNext) THEN
		IF SIf.intCmd = stStateMachine.intState THEN
			SIf.intCmd := cRFD_CMD_DONE;
		END_IF
	END_IF
END_METHOD

METHOD PROTECTED sta_WaitForJob : BOOL
// state implemetation
//--------------------------------------------------------------------------------------
// Entry action
	IF (stStateMachine.intState<>stStateMachine.intStateLastCycle) THEN
		stStateMachine.intStateLastCycle := stStateMachine.intState;
		
	END_IF


//--------------------------------------------------------------------------------------
// Cyclic action
	IF (stStateMachine.intState=stStateMachine.intStateLastCycle) THEN

		
		// State Change Condition
		IF (FALSE) THEN
			stStateMachine.intStateNext := cRFD_STA_Error;
		ELSIF (SIf.intCmd=cRFD_CMD_Read) THEN
			stStateMachine.intStateNext := cRFD_STA_ReadBusy;
		ELSIF (SIf.intCmd=cRFD_CMD_CTRL_ON) THEN
			stStateMachine.intStateNext := cRFD_STA_PowerOnBusy;
		ELSIF (SIf.intCmd=cRFD_CMD_Write) THEN
			stStateMachine.intStateNext := cRFD_STA_WriteBusy;
		ELSIF (SIf.intCmd=cRFD_CMD_MDS) THEN
			stStateMachine.intStateNext := cRFD_STA_MDSBusy;
		ELSIF (SIf.intCmd=cRFD_CMD_SLG) THEN
			stStateMachine.intStateNext := cRFD_STA_SLGBusy;
		ELSIF (SIf.intCmd=cRFD_CMD_CTRL_OFF) THEN
			stStateMachine.intStateNext := cRFD_STA_OFFBusy;
		ELSIF (SIf.intCmd=cRFD_STA_CheckBusy) THEN
			stStateMachine.intStateNext := cRFD_STA_CheckBusy;
		END_IF
		
	END_IF

//--------------------------------------------------------------------------------------
// Exit action
	IF (stStateMachine.intState<>stStateMachine.intStateNext) THEN
		;
	END_IF
END_METHOD

METHOD PROTECTED sta_WriteBusy : BOOL
// state implemetation
//--------------------------------------------------------------------------------------
// Entry action
	IF (stStateMachine.intState<>stStateMachine.intStateLastCycle) THEN
			stStateMachine.intStateLastCycle := stStateMachine.intState;
			// Byte 0 => Lenght
			aTxData[0] := 5 + SIf.stCur.usiCount;
			// Byte 1 => Command write 1=single; 11=continious
			aTxData[1] := 1;
			// Byte 2 => Spare
			aTxData[2] := 0;
			// Byte 3 => Adress MSB
			uinValue := SIf.stCur.uinAdressTag;
			uinValue := ROL(uinValue,8);
			aTxData[3] := UINT_TO_USINT(uinValue);
			// Byte 4 => Adress LSB
			aTxData[4] := UINT_TO_USINT(SIf.stCur.uinAdressTag);
			// Byte 5 =>Lenght
			aTxData[5] := SIf.stCur.usiCount;
 
			IF ((SIf.stCur.uinAdressData+SIf.stCur.usiCount <= 255) AND (SIf.stCur.usiCount+6 <= 255)) THEN
				FOR udiLoopBuffer := 0 TO (SIf.stCur.usiCount) DO
					aTxData[udiLoopBuffer+6] := SIf.stCur.pData^[SIf.stCur.uinAdressData+udiLoopBuffer];
				END_FOR	
				udiComSizeSendData := SIf.stCur.usiCount+6;
				bolComSend := TRUE;		
			ELSE
				SIf.stErr.bolComError := TRUE;
			END_IF
							
	END_IF


//--------------------------------------------------------------------------------------
// Cyclic action
	IF (stStateMachine.intState=stStateMachine.intStateLastCycle) THEN
		
		// State Change Condition
		IF (SIf.stErr.bolComError = TRUE) OR ((SIf.stErr.bolRFIDError = TRUE) AND (udiJobCount > SIf.stCfg.udiRetry)) THEN
			stStateMachine.intStateNext := cRFD_STA_Error;
		ELSIF (SIf.stErr.bolRFIDError = TRUE) THEN
			udiJobCount := udiJobCount + 1;
			stStateMachine.intStateLastCycle := 0; // Startcycle again
		ELSIF ((SIf.stErr.bolComError = 0) AND (bolWriteDone = TRUE)) THEN
			bolWriteDone := FALSE;
			udiJobCount := 0;
			stStateMachine.intStateNext := cRFD_STA_WaitForJob;
		END_IF
	
	END_IF

//--------------------------------------------------------------------------------------
// Exit action
	IF (stStateMachine.intState<>stStateMachine.intStateNext) THEN
		SIf.intCmd := cRFD_CMD_DONE;
	END_IF
END_METHOD

METHOD PROTECTED StateMachine : BOOL

// main statemachine of base controller
CASE stStateMachine.intState OF
	cRFD_STA_OffBusy: 
        THIS^.sta_OffBusy();
	cRFD_STA_Off: 
        THIS^.sta_Off();
    cRFD_STA_PowerOnBusy: 
        THIS^.sta_PowerOnBusy();
	cRFD_STA_WaitForJob: 
        THIS^.sta_WaitForJob();
	cRFD_STA_WriteBusy: 
        THIS^.sta_WriteBusy();
    cRFD_STA_ReadBusy: 
        THIS^.sta_ReadBusy();
	cRFD_STA_TagInitBusy: 
        THIS^.sta_TagInitBusy();
	cRFD_STA_CheckBusy: 
        THIS^.sta_CheckBusy();
	cRFD_STA_MDSBusy: 
        THIS^.sta_MDSBusy();
	cRFD_STA_SLGBusy: 
        THIS^.sta_SLGBusy();
    cRFD_STA_Error: 
        THIS^.sta_Error();
END_CASE;
END_METHOD

METHOD PROTECTED StateMachine_Service : BOOL


// main statemachine of base controller
CASE SIf.intServiceCmd OF
//	cRFD_CMD_MDS: 
//		THIS^.sJobWriteParameter();
//	cYAD_SCMD_READ_PARA: 
//		THIS^.sJobReadParameter();
//	cYAD_SCMD_RESET_ABSENCODER: 
//		THIS^.sJobAbsEncReset();
ELSE
	usiCaseScmd := 0;
	

	
END_CASE;
END_METHOD

END_FUNCTION_BLOCK

// POUs/Controller/Driver/RFD (RFID Driver)/FB_RFR
FUNCTION_BLOCK FB_RFR
VAR
	bolActivate: BOOL := TRUE;
	bolInitDone: BOOL;
	bolInitComDone: BOOL;
	///Communication sending is busy to the serial Card
	bolComSend: BOOL;
	/// Size of Sendingdata
	udiComSizeSendData: UDINT;
	///Communication Data Received
	bolComDataReceived: BOOL;
	/// Size of received Data from serial interface
	udiComSizeReceiveData: UDINT;
	///Sdo Setting is busy to the serial Card
	bolSdoBusy: BOOL;
	///Sdo Setting executing
	bolSdoExecute: BOOL;
	/// Job Reading is done
	bolReadDone: BOOL;
	/// Job Writing is done
	bolWriteDone: BOOL;
	/// Job Reset SLG is done
	bolResetJobDone: BOOL;
	/// Job Reset SLG has Error
	bolResetJobError: BOOL;
	/// Information to SDO Error
	udiSdoErrorNbr: UDINT;
	/// Information to Error
	udiComErrorNbr: UDINT;
	/// Count Reset cycles
	udiResetCount: UDINT;
	/// Count Job Tryals
	udiJobCount: UDINT;
	/// State information from RF ID Tag
	bytRFIDState: BYTE;
	/// BCC Calculation
	bytCheckValue: BYTE;
	/// driver specific interface
	SIf: T_RFD;
	/// get direct Buffer from Interface
	/// access over mapping!! {attribute 'TcLinkTo':='TIID^Device 1 (EtherCAT)^Box 1 (SGDV-E1 CoE Drive)^2nd Transmit PDO mapping^Status word'}
	aRxData: ARRAY[0..255] OF BYTE;
	aTxData: ARRAY[0..255] OF BYTE;
	/// Function for serial communication
	fbEcCoeSdoWrite: TC2_ETHERCAT.FB_EcCoESdoWrite;
	fbExCom: FB_ExCom;
	stStateMachine: T_RFD_StateMachine;
	stSubStateMachine: T_RFD_StateMachine;
	///case variable
	usiCase: USINT;
	///case variable for service cmd's
	usiCaseScmd: USINT;
	/// help values for parameter handling
	sinValue: SINT;
	intValue: INT;
	dinValue: DINT;
	usiValue: USINT;
	uinValue: UINT;
	udiValue: UDINT;
	uliValue: ULINT;
	pTemp: POINTER TO ARRAY[0..7] OF BYTE;
	strTemp: STRING(18);
	udiI: UDINT;
	udiLoopBuffer: UDINT;
	udiLoopData: UDINT;
	udiLoopSend: UDINT;
END_VAR

(*__________________________________________________________________________________________________
¦	
¦	Vistaprint Schweiz GmbH
¦	CH - 8401 Winterthur
¦
¦	www.vistaprint.ch - info@vistaprint.ch
¦___________________________________________________________________________________________________

Function desription:
Driver for Simatic RFID Reader RF382R 6GT2801-3AB20-0AX0 (only read function)


History:
Version		Date			Author		Comment
---------------------------------------------------------------------------------------------------
0.00.1		09.07.2013		AVME/PRE	Start history
0.00.2		18.09.2013		AVME/KVO	no initial write of parameter to RFID reader at PowerOnBusy
0.00.3		25.09.2013		AVME/KVO	always set sample error and go to error state!
___________________________________________________________________________________________________*)


IF (bolActivate) THEN // cyclic call enabled
	
	IF (bolInitDone=FALSE) THEN // first cycle -> init
		CtrlInit();
		bolInitDone := TRUE;
	ELSE
		CycleStartDuty();
		
		StateMachine_Service(); // handles asynchron service commands
		
		StateMachine();
		
		CycleEndDuty();
	END_IF
	
END_IF;

METHOD PROTECTED CtrlInit : BOOL
// one time first cyclic call
;
END_METHOD

METHOD PROTECTED CycleEndDuty : BOOL
SIf.strState := THIS^.getCmdState(intCmdState:=stStateMachine.intState,bolState:=TRUE);

IF (stStateMachine.intState<>stStateMachine.intStateNext) THEN
	stStateMachine.intState := stStateMachine.intStateNext;  // set next state for next cycle
END_IF

(***************************************************************
        Function Block Calls
***************************************************************)
END_METHOD

METHOD PROTECTED CycleStartDuty : BOOL
// ----------------------------------------------------------------------------------
// cyclic actions outside of statemachine
fbExCom(
	In_pRxData:= ADR(aRxData), 
	In_pTxData:= ADR(aTxData), 
	In_udiTxCount:= udiComSizeSendData, 
	In_bolErrorAck:= SIf.stErr.bolErrAck, 
	InOut_bolSend:= bolComSend, 
	InOut_bolRec:= bolComDataReceived, 
	Out_udiRxCount=> udiComSizeReceiveData, 
	Out_bolComError=> SIf.stErr.bolComError, 
	Out_bolProtocolErr=> SIf.stErr.bolProtcolError, 
	Out_udiErrorCode=> udiComErrorNbr);

(* program code at the beginning of each PLC cycle *)
IF bolInitComDone=TRUE THEN
	// Received Data checking and interpreting
	IF bolComDataReceived = TRUE THEN
		IF (aRxData[0] = 1) AND (udiComSizeReceiveData = 3) THEN		// Ack Reset
			IF aRxData[1] = 0 THEN
				bolResetJobDone := TRUE;
			ELSE
				 SIf.stErr.bolProtcolError := TRUE;
			END_IF
		ELSE
			// UID
			MEMCPY(destAddr:=ADR(strTemp), srcAddr:=ADR(aRxData[0]), n:=16);

			uliValue := FB_HEXSTRING_TO_ULINT(in_strSTRING:= strTemp);
			pTemp := ADR(SIf.stStatus.abyteUID[0]);
			MEMCPY(destAddr:=ADR(SIf.stStatus.abyteUID[0]), srcAddr:=ADR(uliValue), n:=8);		// COPY to ID 
			
		END_IF
		bolComDataReceived := FALSE;
	END_IF
END_IF

// always go to Error 
IF ((SIf.stErr.bolProtcolError) OR  (SIf.stErr.bolRFIDError) OR (SIf.stErr.bolSDOError)) THEN
	SIf.stErr.bolErrorActive := TRUE; // set sample Error -> got to Error state
END_IF

IF (SIf.stErr.bolErrorActive) AND (stStateMachine.intState<>cRFD_STA_Error)  THEN
	stStateMachine.intStateNext := cRFD_STA_Error;
ELSIF (stStateMachine.intState<cRFD_STA_PowerOnBusy) AND (stStateMachine.intState<>cRFD_STA_Error) THEN
	stStateMachine.intStateNext := cRFD_STA_PowerOnBusy;
END_IF

SIf.strCmd := THIS^.getCmdState(intCmdState:=SIf.intCmd,bolState:=FALSE);
END_METHOD

METHOD FB_init : BOOL
VAR_INPUT
	///if TRUE, the retain variables are initialized (warm start / cold start)
	bInitRetains: BOOL;
	///if TRUE, the instance afterwards gets moved into the copy code (online change)
	bInCopyCode: BOOL;
END_VAR
VAR
	udiTaskCnt: UDINT;
	ii: UINT;
END_VAR
SIf.intCmd := cRFD_CMD_DONE;
SIf.intServiceCmd := cRFD_CMD_DONE; // not used at the moment
stStateMachine.intStateLastCycle  := cRFD_CMD_DONE; //EntryStop of power BASE_PLC.OFF enable

// Communication Settings
SIf.stCfg.eTyp := E_Typ_RFW.RF382R;
SIf.stCfg.uinBaudrate := UINT_TO_USINT(E_Typ_Baudrate.baud_38400);
SIf.stCfg.stNetId := '192.168.70.26.3.1';
SIf.stCfg.uinSlaveAddr := 1002;
END_METHOD

METHOD PROTECTED getCmdState : STRING
VAR_INPUT
	intCmdState: INT;
	bolState: BOOL;
END_VAR
// get string cmd/state string information in runtime
IF (bolState=FALSE) THEN
	// cmd's
	CASE intCmdState OF
		cRFD_CMD_DONE: 
			getCmdState := 'cRFD_CMD_DONE';
		cRFD_CMD_CTRL_ON: 
			getCmdState := 'cRFD_CMD_CTRL_ON';

	END_CASE;
ELSE

// States
	CASE intCmdState OF
		cRFD_STA_Error: 
			getCmdState := 'cRFD_STA_Error';
		cRFD_STA_WaitForJob: 
			getCmdState := 'cRFD_STA_WaitForJob';
		cRFD_STA_PowerOnBusy: 
			getCmdState := 'cRFD_STA_PowerOnBusy';

	END_CASE;
END_IF
END_METHOD

METHOD getSIf : POINTER TO T_RFD
getSIf := ADR(SIf);
END_METHOD

METHOD PROTECTED sta_Error : BOOL
// state implemetation
//--------------------------------------------------------------------------------------
// Entry action
	IF (stStateMachine.intState<>stStateMachine.intStateLastCycle) THEN
		stStateMachine.intStateHistory := stStateMachine.intStateLastCycle;
		stStateMachine.intStateLastCycle := stStateMachine.intState;
		
	END_IF


//--------------------------------------------------------------------------------------
// Cyclic action
	IF (stStateMachine.intState=stStateMachine.intStateLastCycle) THEN
		SIf.stErr.bolErrorActive := TRUE;
		IF (SIf.stErr.bolComError = TRUE) OR (SIf.stErr.bolProtcolError = TRUE) THEN
			SIf.stErr.udiErrorID := udiComErrorNbr;
		ELSIF SIf.stErr.bolSDOError = TRUE THEN
			SIf.stErr.udiErrorID := udiSdoErrorNbr;
		ELSIF (udiResetCount >=SIf.stCfg.udiRetry) OR (udiJobCount >= SIf.stCfg.udiRetry) THEN
			SIf.stErr.udiErrorID := SIf.stCfg.udiRetry;
		ELSE
			SIf.stErr.udiErrorID := 0;
		END_IF

		
		// State Change Condition
		IF (SIf.stErr.bolErrAck = TRUE) THEN
			// Reset all active errors
			SIf.stErr.bolErrorActive := FALSE;
			SIf.stErr.bolComError := FALSE;
			SIf.stErr.bolProtcolError := FALSE;
			SIf.stErr.bolSDOError := FALSE;
			SIf.stErr.udiErrorID := 0;
			stStateMachine.intStateNext := cRFD_STA_PowerOnBusy;		
		END_IF
	END_IF




//--------------------------------------------------------------------------------------
// Exit action
	IF (stStateMachine.intState<>stStateMachine.intStateNext) THEN
		;
	END_IF
END_METHOD

METHOD PROTECTED sta_PowerOnBusy : BOOL
// state implemetation
//--------------------------------------------------------------------------------------
// Entry action
	IF (stStateMachine.intState<>stStateMachine.intStateLastCycle) THEN
		stStateMachine.intStateLastCycle := stStateMachine.intState;
			//IF bolInitComDone=FALSE THEN
				// direct write parameter doesn't work!! KVO 17.09.2013 with new Kannegiesser RFID
				// Feedback rx[0..2] 255 4 251 -> Baudrate/task time not 2ms
				// no Feedback -> parameter set? estimated  rx[0..2] 1 0 1
				// decision with Rolf Engelputzeder 18.09.2013 
				// don't use write parameter at the moment:
				stSubStateMachine.intState := cRFD_SUB_SubStatesEnd;// cRFD_SUB_ClearBuffer;		// First Time set Baudrate and communication Settings
				stSubStateMachine.intStateNext := cRFD_SUB_SubStatesEnd;// cRFD_SUB_ClearBuffer;		// First Time set Baudrate and communication Settings
				bolInitComDone := TRUE; // old without this condition
				
				(*
				// original set parameter to RFID
				stSubStateMachine.intState := cRFD_SUB_ClearBuffer;		// First Time set Baudrate and communication Settings
				stSubStateMachine.intStateNext := cRFD_SUB_ClearBuffer;
				*)
			//END_IF
			bolSdoExecute := FALSE;
			bolResetJobDone := FALSE;
	END_IF


//--------------------------------------------------------------------------------------
// Cyclic action
	IF (stStateMachine.intState=stStateMachine.intStateLastCycle) THEN
		
		// main statemachine of base controller
		CASE stSubStateMachine.intState OF
			cRFD_SUB_SetBaudrate:
				IF stSubStateMachine.intStateLastCycle <> stSubStateMachine.intState THEN
					stSubStateMachine.intStateLastCycle := stSubStateMachine.intState;
				END_IF
				fbEcCoeSdoWrite(
					sNetId:= SIf.stCfg.stNetId, 
					nSlaveAddr:= SIf.stCfg.uinSlaveAddr, 
					nIndex:= SIf.stCfg.uinCoeIndexComSettings, 
					nSubIndex:= SIf.stCfg.usiCoeSubindexComBaudrate, 
					pSrcBuf:= ADR(SIf.stCfg.uinBaudrate), 
					cbBufLen:= SIZEOF(SIf.stCfg.uinBaudrate), 
					bExecute:= bolSdoExecute, 
					tTimeout:= DEFAULT_ADS_TIMEOUT, 
					bBusy=> bolSdoBusy, 
					bError=> SIf.stErr.bolSDOError, 
					nErrId=> udiSdoErrorNbr);
					
					
				IF 	(bolSdoExecute = TRUE) THEN
					IF ((SIf.stErr.bolSDOError = FALSE) AND (bolSdoBusy = FALSE)) THEN
						bolSdoExecute := FALSE;
						stSubStateMachine.intStateNext := cRFD_SUB_ClearBuffer;
					END_IF
				ELSE
					bolSdoExecute := TRUE;
				END_IF
				
			
			cRFD_SUB_SetComSettings:
				IF stSubStateMachine.intStateLastCycle <> stSubStateMachine.intState THEN
					stSubStateMachine.intStateLastCycle := stSubStateMachine.intState;
				END_IF
				fbEcCoeSdoWrite(
					sNetId:= SIf.stCfg.stNetId, 
					nSlaveAddr:= SIf.stCfg.uinSlaveAddr, 
					nSubIndex:= SIf.stCfg.usiCoeSubindexComDataframe, 
					nIndex:= SIf.stCfg.uinCoeIndexComSettings, 
					pSrcBuf:= ADR(SIf.stCfg.uinComSettings), 
					cbBufLen:= SIZEOF(SIf.stCfg.uinComSettings), 
					bExecute:= bolSdoExecute, 
					tTimeout:= T#2S, 
					bBusy=> bolSdoBusy, 
					bError=> SIf.stErr.bolSDOError, 
					nErrId=> udiSdoErrorNbr);
					
				IF 	(bolSdoExecute = TRUE) THEN
					IF ((SIf.stErr.bolSDOError = FALSE) AND (bolSdoBusy = FALSE)) THEN
						bolSdoExecute := FALSE;
						stSubStateMachine.intStateNext := cRFD_SUB_ClearBuffer;
					END_IF
				ELSE
					bolSdoExecute := TRUE;
				END_IF

	
			cRFD_SUB_ClearBuffer: 	 
				IF stSubStateMachine.intStateLastCycle <> stSubStateMachine.intState THEN
					stSubStateMachine.intStateLastCycle := stSubStateMachine.intState;
				END_IF
				bolInitComDone := TRUE;
				IF (SIf.stErr.bolComError = FALSE) THEN
					stSubStateMachine.intStateNext := cRFD_SUB_InitString;
				END_IF

				
			cRFD_SUB_InitString: 
				IF stSubStateMachine.intStateLastCycle <> stSubStateMachine.intState THEN
					stSubStateMachine.intStateLastCycle := stSubStateMachine.intState;
					// Byte 0 => Para = 16#01
					aTxData[0] := 1;
					// Byte 1 => Memory
					aTxData[1] := SIf.stCfg.usiMemory;
					// Byte 2 => Spare
					aTxData[2] := 0;
					// Byte 3 => Spare
					aTxData[3] := 0;
					// Byte 4 => Spare
					aTxData[4] := 0;
					// Byte 5 => Spare
					aTxData[5] := 0;
					// Byte 6 => Spare
					aTxData[6] := 0;
					// Byte 7 => Scan Mode
					aTxData[7] := SIf.stCfg.usiScanMode;
					// Byte 8 => Lock Time High Byte
					aTxData[8] := UINT_TO_BYTE(SIf.stCfg.uinLockTime_ms/100);
					// Byte 9 => Lock Time Low Byte
					aTxData[9] := UINT_TO_BYTE(SHR((SIf.stCfg.uinLockTime_ms/100),8));
					// Byte 10 => Spare
					aTxData[10] := 0;
					// Byte 11 => Spare
					aTxData[11] := 0;
					// Byte 12 => Spare
					aTxData[12] := 0;
					// Byte 13 => Spare
					aTxData[13] := 0;
					// Byte 14 => Spare
					aTxData[14] := 0;
					// Byte 15 => Spare
					aTxData[15] := 0;
					// Byte 16 => Spare
					aTxData[16] := 0;
					// Byte 17 => Spare
					aTxData[17] := 0;
					// Byte 18 => Spare
					aTxData[18] := 0;
					// Byte 19 => Spare
					aTxData[19] := 0;
					// Byte 20 => Spare
					aTxData[20] := 0;
					// Byte 21 => Spare
					aTxData[21] := 0;
					// Byte 22 => Spare
					aTxData[22] := 0;

					bytCheckValue := aTxData[0] XOR aTxData[1];
					FOR udiI := 2 TO  22 DO
						bytCheckValue := bytCheckValue XOR aTxData[udiI];
					END_FOR
					
					// Byte 23 => BCC
					aTxData[23] := bytCheckValue;
					
					udiComSizeSendData := 24;
					bolComSend := TRUE;
				END_IF
			
